gfCNCPoint4[8472] = {X 422.2320, Y 54.5599, Z -5.5000, A 0.000, B 0.000, C 0.000 }
gfCNCPoint4[8473] = {X 422.9287, Y 55.2566, Z -5.5000, A 0.000, B 0.000, C 0.000 }
gfCNCPoint4[8474] = {X 423.4529, Y 56.0909, Z -5.5000, A 0.000, B 0.000, C 0.000 }
gfCNCPoint4[8475] = {X 423.7783, Y 57.0209, Z -5.5000, A 0.000, B 0.000, C 0.000 }
gfCNCPoint4[8476] = {X 423.8886, Y 58.0000, Z -5.5000, A 0.000, B 0.000, C 0.000 }
gfCNCPoint4[8477] = {X 423.8886, Y 58.1773, Z -5.5000, A 0.000, B 0.000, C 0.000 }
gfCNCPoint4[8478] = {X 429.6420, Y 60.4190, Z -5.5000, A 0.000, B 0.000, C 0.000 }
gfCNCPoint4[8479] = {X 457.7784, Y 71.5825, Z -5.5000, A 0.000, B 0.000, C 0.000 }
gfCNCPoint4[8480] = {X 457.7788, Y 63.2811, Z -5.5000, A 0.000, B 0.000, C 0.000 }
gfCNCPoint4[8481] = {X 456.9197, Y 63.0558, Z -5.5000, A 0.000, B 0.000, C 0.000 }
gfCNCPoint4[8482] = {X 456.1233, Y 62.6625, Z -5.5000, A 0.000, B 0.000, C 0.000 }
gfCNCPoint4[8483] = {X 455.4221, Y 62.1174, Z -5.5000, A 0.000, B 0.000, C 0.000 }
gfCNCPoint4[8484] = {X 454.8446, Y 61.4425, Z -5.5000, A 0.000, B 0.000, C 0.000 }
gfCNCPoint4[8485] = {X 454.4145, Y 60.6654, Z -5.5000, A 0.000, B 0.000, C 0.000 }
gfCNCPoint4[8486] = {X 454.1492, Y 59.8177, Z -5.5000, A 0.000, B 0.000, C 0.000 }
gfCNCPoint4[8487] = {X 454.0596, Y 58.9341, Z -5.5000, A 0.000, B 0.000, C 0.000 }
gfCNCPoint4[8488] = {X 454.0596, Y 58.0000, Z -5.5000, A 0.000, B 0.000, C 0.000 }
gfCNCPoint4[8489] = {X 454.1699, Y 57.0209, Z -5.5000, A 0.000, B 0.000, C 0.000 }
gfCNCPoint4[8490] = {X 454.4953, Y 56.0909, Z -5.5000, A 0.000, B 0.000, C 0.000 }
gfCNCPoint4[8491] = {X 455.0195, Y 55.2566, Z -5.5000, A 0.000, B 0.000, C 0.000 }
gfCNCPoint4[8492] = {X 455.7162, Y 54.5599, Z -5.5000, A 0.000, B 0.000, C 0.000 }
gfCNCPoint4[8493] = {X 456.5505, Y 54.0357, Z -5.5000, A 0.000, B 0.000, C 0.000 }
gfCNCPoint4[8494] = {X 457.4805, Y 53.7103, Z -5.5000, A 0.000, B 0.000, C 0.000 }
gfCNCPoint4[8495] = {X 458.4596, Y 53.6000, Z -5.5000, A 0.000, B 0.000, C 0.000 }
gfCNCPoint4[8496] = {X 475.0000, Y 53.6000, Z -5.5000, A 0.000, B 0.000, C 0.000 }
gfCNCPoint4[8497] = {X 475.9791, Y 53.7103, Z -5.5000, A 0.000, B 0.000, C 0.000 }
gfCNCPoint4[8498] = {X 476.9091, Y 54.0357, Z -5.5000, A 0.000, B 0.000, C 0.000 }
gfCNCPoint4[8499] = {X 477.7434, Y 54.5599, Z -5.5000, A 0.000, B 0.000, C 0.000 }
gfCNCPoint4[8500] = {X 478.4401, Y 55.2566, Z -5.5000, A 0.000, B 0.000, C 0.000 }
gfCNCPoint4[8501] = {X 478.9643, Y 56.0909, Z -5.5000, A 0.000, B 0.000, C 0.000 }
gfCNCPoint4[8502] = {X 479.2897, Y 57.0209, Z -5.5000, A 0.000, B 0.000, C 0.000 }
gfCNCPoint4[8503] = {X 479.4000, Y 58.0000, Z -5.5000, A 0.000, B 0.000, C 0.000 }
gfCNCPoint4[8504] = {X 479.3998, Y 58.9704, Z -5.5000, A 0.000, B 0.000, C 0.000 }
gfCNCPoint4[8505] = {X 479.3040, Y 59.8483, Z -5.5000, A 0.000, B 0.000, C 0.000 }
gfCNCPoint4[8506] = {X 479.0347, Y 60.6893, Z -5.5000, A 0.000, B 0.000, C 0.000 }
gfCNCPoint4[8507] = {X 478.6030, Y 61.4596, Z -5.5000, A 0.000, B 0.000, C 0.000 }
gfCNCPoint4[8508] = {X 478.0261, Y 62.1282, Z -5.5000, A 0.000, B 0.000, C 0.000 }
gfCNCPoint4[8509] = {X 477.3273, Y 62.6682, Z -5.5000, A 0.000, B 0.000, C 0.000 }
gfCNCPoint4[8510] = {X 476.5348, Y 63.0577, Z -5.5000, A 0.000, B 0.000, C 0.000 }
gfCNCPoint4[8511] = {X 475.6805, Y 63.2811, Z -5.5000, A 0.000, B 0.000, C 0.000 }
gfCNCPoint4[8512] = {X 475.6809, Y 92.7040, Z -5.5000, A 0.000, B 0.000, C 0.000 }
gfCNCPoint4[8513] = {X 476.0501, Y 92.7986, Z -5.5000, A 0.000, B 0.000, C 0.000 }
gfCNCPoint4[8514] = {X 476.4143, Y 92.9108, Z -5.5000, A 0.000, B 0.000, C 0.000 }
gfCNCPoint4[8515] = {X 477.2408, Y 93.2866, Z -5.5000, A 0.000, B 0.000, C 0.000 }
gfCNCPoint4[8516] = {X 477.9718, Y 93.8249, Z -5.5000, A 0.000, B 0.000, C 0.000 }
gfCNCPoint4[8517] = {X 478.5759, Y 94.5026, Z -5.5000, A 0.000, B 0.000, C 0.000 }
gfCNCPoint4[8518] = {X 479.0270, Y 95.2905, Z -5.5000, A 0.000, B 0.000, C 0.000 }
gfCNCPoint4[8519] = {X 479.3057, Y 96.1545, Z -5.5000, A 0.000, B 0.000, C 0.000 }
gfCNCPoint4[8520] = {X 479.4000, Y 97.0575, Z -5.5000, A 0.000, B 0.000, C 0.000 }
gfCNCPoint4[8521] = {X 479.4000, Y 97.6951, Z -5.5000, A 0.000, B 0.000, C 0.000 }
gfCNCPoint4[8522] = {X 479.8800, Y 97.6951, Z -5.5000, A 0.000, B 0.000, C 0.000 }
gfCNCPoint4[8523] = {X 507.6814, Y 97.6951, Z -5.5000, A 0.000, B 0.000, C 0.000 }
gfCNCPoint4[8524] = {X 507.6814, Y 100.0951, Z -5.5000, A 0.000, B 0.000, C 0.000 }
gfCNCPoint4[8525] = {X 600.0148, Y 100.0951, Z -5.5000, A 0.000, B 0.000, C 0.000 }
gfCNCPoint4[8526] = {X 600.0672, Y 100.0698, Z -5.5000, A 0.000, B 0.000, C 0.000 }
gfCNCPoint4[8527] = {X 600.0949, Y 100.0187, Z -5.5000, A 0.000, B 0.000, C 0.000 }
gfCNCPoint4[8528] = {X 600.0966, Y 99.1432, Z -5.5000, A 0.000, B 0.000, C 0.000 }
gfCNCPoint4[8529] = {X 600.0966, Y 49.8790, Z -5.5000, A 0.000, B 0.000, C 0.000 }
gfCNCPoint4[8530] = {X 601.1112, Y 49.7518, Z -5.5000, A 0.000, B 0.000, C 0.000 }
gfCNCPoint4[8531] = {X 602.0770, Y 49.4159, Z -5.5000, A 0.000, B 0.000, C 0.000 }
gfCNCPoint4[8532] = {X 602.9516, Y 48.8862, Z -5.5000, A 0.000, B 0.000, C 0.000 }
gfCNCPoint4[8533] = {X 603.6966, Y 48.1858, Z -5.5000, A 0.000, B 0.000, C 0.000 }
gfCNCPoint4[8534] = {X 603.6966, Y 47.3864, Z -5.5000, A 0.000, B 0.000, C 0.000 }
gfCNCPoint4[8535] = {X 603.1503, Y 48.0717, Z -5.5000, A 0.000, B 0.000, C 0.000 }
gfCNCPoint4[8536] = {X 602.4791, Y 48.6351, Z -5.5000, A 0.000, B 0.000, C 0.000 }
gfCNCPoint4[8537] = {X 601.7094, Y 49.0544, Z -5.5000, A 0.000, B 0.000, C 0.000 }
gfCNCPoint4[8538] = {X 600.8720, Y 49.3127, Z -5.5000, A 0.000, B 0.000, C 0.000 }
gfCNCPoint4[8539] = {X 600.0000, Y 49.4000, Z -5.5000, A 0.000, B 0.000, C 0.000 }
gfCNCPoint4[8540] = {X 593.5565, Y 49.4000, Z -5.5000, A 0.000, B 0.000, C 0.000 }
gfCNCPoint4[8541] = {X 592.5988, Y 49.2945, Z -5.5000, A 0.000, B 0.000, C 0.000 }
gfCNCPoint4[8542] = {X 591.6870, Y 48.9831, Z -5.5000, A 0.000, B 0.000, C 0.000 }
gfCNCPoint4[8543] = {X 590.8648, Y 48.4806, Z -5.5000, A 0.000, B 0.000, C 0.000 }
gfCNCPoint4[8544] = {X 590.1717, Y 47.8112, Z -5.5000, A 0.000, B 0.000, C 0.000 }
gfCNCPoint4[8545] = {X 589.6410, Y 47.0071, Z -5.5000, A 0.000, B 0.000, C 0.000 }
gfCNCPoint4[8546] = {X 589.3741, Y 46.3664, Z -5.5000, A 0.000, B 0.000, C 0.000 }
gfCNCPoint4[8547] = {X 589.2113, Y 45.6918, Z -5.5000, A 0.000, B 0.000, C 0.000 }
gfCNCPoint4[8548] = {X 589.1565, Y 45.0000, Z -5.5000, A 0.000, B 0.000, C 0.000 }
gfCNCPoint4[8549] = {X 589.1565, Y 44.0643, Z -5.5000, A 0.000, B 0.000, C 0.000 }
gfCNCPoint4[8550] = {X 589.2606, Y 43.1278, Z -5.5000, A 0.000, B 0.000, C 0.000 }
gfCNCPoint4[8551] = {X 589.5599, Y 42.2344, Z -5.5000, A 0.000, B 0.000, C 0.000 }
gfCNCPoint4[8552] = {X 590.0411, Y 41.4243, Z -5.5000, A 0.000, B 0.000, C 0.000 }
gfCNCPoint4[8553] = {X 590.6824, Y 40.7340, Z -5.5000, A 0.000, B 0.000, C 0.000 }
gfCNCPoint4[8554] = {X 590.6838, Y 40.3070, Z -5.5000, A 0.000, B 0.000, C 0.000 }
gfCNCPoint4[8555] = {X 590.6830, Y 35.2188, Z -5.5000, A 0.000, B 0.000, C 0.000 }
gfCNCPoint4[8556] = {X 590.6828, Y 33.9412, Z -5.5000, A 0.000, B 0.000, C 0.000 }
gfCNCPoint4[8557] = {X 585.5192, Y 46.6830, Z -5.5000, A 0.000, B 0.000, C 0.000 }
gfCNCPoint4[8558] = {X 585.4476, Y 46.8466, Z -5.5000, A 0.000, B 0.000, C 0.000 }
gfCNCPoint4[8559] = {X 585.3694, Y 47.0071, Z -5.5000, A 0.000, B 0.000, C 0.000 }
gfCNCPoint4[8560] = {X 584.8417, Y 47.8075, Z -5.5000, A 0.000, B 0.000, C 0.000 }
gfCNCPoint4[8561] = {X 584.1532, Y 48.4747, Z -5.5000, A 0.000, B 0.000, C 0.000 }
gfCNCPoint4[8562] = {X 583.3365, Y 48.9769, Z -5.5000, A 0.000, B 0.000, C 0.000 }
gfCNCPoint4[8563] = {X 582.4111, Y 49.2946, Z -5.5000, A 0.000, B 0.000, C 0.000 }
gfCNCPoint4[8564] = {X 581.4384, Y 49.4000, Z -5.5000, A 0.000, B 0.000, C 0.000 }
gfCNCPoint4[8565] = {X 580.4664, Y 49.2878, Z -5.5000, A 0.000, B 0.000, C 0.000 }
gfCNCPoint4[8566] = {X 579.5433, Y 48.9635, Z -5.5000, A 0.000, B 0.000, C 0.000 }
gfCNCPoint4[8567] = {X 578.7146, Y 48.4433, Z -5.5000, A 0.000, B 0.000, C 0.000 }
gfCNCPoint4[8568] = {X 578.0214, Y 47.7529, Z -5.5000, A 0.000, B 0.000, C 0.000 }
gfCNCPoint4[8569] = {X 577.4979, Y 46.9263, Z -5.5000, A 0.000, B 0.000, C 0.000 }
gfCNCPoint4[8570] = {X 577.4375, Y 46.7968, Z -5.5000, A 0.000, B 0.000, C 0.000 }
gfCNCPoint4[8571] = {X 577.3813, Y 46.6655, Z -5.5000, A 0.000, B 0.000, C 0.000 }
gfCNCPoint4[8572] = {X 572.5793, Y 34.9232, Z -5.5000, A 0.000, B 0.000, C 0.000 }
gfCNCPoint4[8573] = {X 572.0992, Y 33.7494, Z -5.5000, A 0.000, B 0.000, C 0.000 }
gfCNCPoint4[8574] = {X 572.0993, Y 35.0176, Z -5.5000, A 0.000, B 0.000, C 0.000 }
gfCNCPoint4[8575] = {X 572.0995, Y 40.7335, Z -5.5000, A 0.000, B 0.000, C 0.000 }
gfCNCPoint4[8576] = {X 572.7439, Y 41.4225, Z -5.5000, A 0.000, B 0.000, C 0.000 }
gfCNCPoint4[8577] = {X 573.2265, Y 42.2331, Z -5.5000, A 0.000, B 0.000, C 0.000 }
gfCNCPoint4[8578] = {X 573.5253, Y 43.1280, Z -5.5000, A 0.000, B 0.000, C 0.000 }
gfCNCPoint4[8579] = {X 573.6264, Y 44.0660, Z -5.5000, A 0.000, B 0.000, C 0.000 }
gfCNCPoint4[8580] = {X 573.6264, Y 45.0000, Z -5.5000, A 0.000, B 0.000, C 0.000 }
gfCNCPoint4[8581] = {X 573.5140, Y 45.9884, Z -5.5000, A 0.000, B 0.000, C 0.000 }
gfCNCPoint4[8582] = {X 573.1824, Y 46.9263, Z -5.5000, A 0.000, B 0.000, C 0.000 }
gfCNCPoint4[8583] = {X 572.6569, Y 47.7553, Z -5.5000, A 0.000, B 0.000, C 0.000 }
gfCNCPoint4[8584] = {X 571.9608, Y 48.4472, Z -5.5000, A 0.000, B 0.000, C 0.000 }
gfCNCPoint4[8585] = {X 571.1286, Y 48.9676, Z -5.5000, A 0.000, B 0.000, C 0.000 }
gfCNCPoint4[8586] = {X 570.2018, Y 49.2905, Z -5.5000, A 0.000, B 0.000, C 0.000 }
gfCNCPoint4[8587] = {X 569.2264, Y 49.4000, Z -5.5000, A 0.000, B 0.000, C 0.000 }
gfCNCPoint4[8588] = {X 562.4443, Y 49.4000, Z -5.5000, A 0.000, B 0.000, C 0.000 }
gfCNCPoint4[8589] = {X 561.4652, Y 49.2897, Z -5.5000, A 0.000, B 0.000, C 0.000 }
gfCNCPoint4[8590] = {X 560.5352, Y 48.9643, Z -5.5000, A 0.000, B 0.000, C 0.000 }
gfCNCPoint4[8591] = {X 559.7009, Y 48.4401, Z -5.5000, A 0.000, B 0.000, C 0.000 }
gfCNCPoint4[8592] = {X 559.0042, Y 47.7434, Z -5.5000, A 0.000, B 0.000, C 0.000 }
gfCNCPoint4[8593] = {X 558.4800, Y 46.9091, Z -5.5000, A 0.000, B 0.000, C 0.000 }
gfCNCPoint4[8594] = {X 558.1546, Y 45.9791, Z -5.5000, A 0.000, B 0.000, C 0.000 }
gfCNCPoint4[8595] = {X 558.0443, Y 45.0000, Z -5.5000, A 0.000, B 0.000, C 0.000 }
gfCNCPoint4[8596] = {X 558.0443, Y 44.0644, Z -5.5000, A 0.000, B 0.000, C 0.000 }
gfCNCPoint4[8597] = {X 558.1481, Y 43.1277, Z -5.5000, A 0.000, B 0.000, C 0.000 }
gfCNCPoint4[8598] = {X 558.4477, Y 42.2341, Z -5.5000, A 0.000, B 0.000, C 0.000 }
gfCNCPoint4[8599] = {X 558.9294, Y 41.4240, Z -5.5000, A 0.000, B 0.000, C 0.000 }
gfCNCPoint4[8600] = {X 559.5715, Y 40.7340, Z -5.5000, A 0.000, B 0.000, C 0.000 }
gfCNCPoint4[8601] = {X 559.5715, Y 9.2668, Z -5.5000, A 0.000, B 0.000, C 0.000 }
gfCNCPoint4[8602] = {X 558.9270, Y 8.5777, Z -5.5000, A 0.000, B 0.000, C 0.000 }
gfCNCPoint4[8603] = {X 558.4443, Y 7.7670, Z -5.5000, A 0.000, B 0.000, C 0.000 }
gfCNCPoint4[8604] = {X 558.1454, Y 6.8720, Z -5.5000, A 0.000, B 0.000, C 0.000 }
gfCNCPoint4[8605] = {X 558.0443, Y 5.9340, Z -5.5000, A 0.000, B 0.000, C 0.000 }
gfCNCPoint4[8606] = {X 558.0443, Y 5.0000, Z -5.5000, A 0.000, B 0.000, C 0.000 }
gfCNCPoint4[8607] = {X 558.1353, Y 4.1096, Z -5.5000, A 0.000, B 0.000, C 0.000 }
gfCNCPoint4[8608] = {X 558.4046, Y 3.2561, Z -5.5000, A 0.000, B 0.000, C 0.000 }
gfCNCPoint4[8609] = {X 558.9155, Y 2.3717, Z -5.5000, A 0.000, B 0.000, C 0.000 }
gfCNCPoint4[8610] = {X 559.6166, Y 1.6289, Z -5.5000, A 0.000, B 0.000, C 0.000 }
gfCNCPoint4[8611] = {X 560.4700, Y 1.0678, Z -5.5000, A 0.000, B 0.000, C 0.000 }
gfCNCPoint4[8612] = {X 561.4298, Y 0.7185, Z -5.5000, A 0.000, B 0.000, C 0.000 }
gfCNCPoint4[8613] = {X 562.4443, Y 0.6000, Z -5.5000, A 0.000, B 0.000, C 0.000 }
gfCNCPoint4[8614] = {X 570.9376, Y 0.6000, Z -5.5000, A 0.000, B 0.000, C 0.000 }
gfCNCPoint4[8615] = {X 571.9520, Y 0.7185, Z -5.5000, A 0.000, B 0.000, C 0.000 }
gfCNCPoint4[8616] = {X 572.9118, Y 1.0678, Z -5.5000, A 0.000, B 0.000, C 0.000 }
gfCNCPoint4[8617] = {X 573.7653, Y 1.6289, Z -5.5000, A 0.000, B 0.000, C 0.000 }
gfCNCPoint4[8618] = {X 574.4663, Y 2.3717, Z -5.5000, A 0.000, B 0.000, C 0.000 }
gfCNCPoint4[8619] = {X 574.9772, Y 3.2561, Z -5.5000, A 0.000, B 0.000, C 0.000 }
gfCNCPoint4[8620] = {X 575.2465, Y 4.1096, Z -5.5000, A 0.000, B 0.000, C 0.000 }
gfCNCPoint4[8621] = {X 575.3376, Y 5.0000, Z -5.5000, A 0.000, B 0.000, C 0.000 }
gfCNCPoint4[8622] = {X 575.3372, Y 5.9910, Z -5.5000, A 0.000, B 0.000, C 0.000 }
gfCNCPoint4[8623] = {X 575.2577, Y 6.7686, Z -5.5000, A 0.000, B 0.000, C 0.000 }
gfCNCPoint4[8624] = {X 575.0418, Y 7.5199, Z -5.5000, A 0.000, B 0.000, C 0.000 }
gfCNCPoint4[8625] = {X 574.6964, Y 8.2211, Z -5.5000, A 0.000, B 0.000, C 0.000 }
gfCNCPoint4[8626] = {X 575.2866, Y 9.6566, Z -5.5000, A 0.000, B 0.000, C 0.000 }
gfCNCPoint4[8627] = {X 581.1912, Y 24.1575, Z -5.5000, A 0.000, B 0.000, C 0.000 }
gfCNCPoint4[8628] = {X 587.7569, Y 8.0998, Z -5.5000, A 0.000, B 0.000, C 0.000 }
gfCNCPoint4[8629] = {X 587.4434, Y 7.4142, Z -5.5000, A 0.000, B 0.000, C 0.000 }
gfCNCPoint4[8630] = {X 587.2515, Y 6.6851, Z -5.5000, A 0.000, B 0.000, C 0.000 }
gfCNCPoint4[8631] = {X 587.1870, Y 5.9340, Z -5.5000, A 0.000, B 0.000, C 0.000 }
gfCNCPoint4[8632] = {X 587.1870, Y 5.0000, Z -5.5000, A 0.000, B 0.000, C 0.000 }
gfCNCPoint4[8633] = {X 587.2780, Y 4.1096, Z -5.5000, A 0.000, B 0.000, C 0.000 }
gfCNCPoint4[8634] = {X 587.5473, Y 3.2561, Z -5.5000, A 0.000, B 0.000, C 0.000 }
gfCNCPoint4[8635] = {X 588.0582, Y 2.3717, Z -5.5000, A 0.000, B 0.000, C 0.000 }
gfCNCPoint4[8636] = {X 588.7592, Y 1.6289, Z -5.5000, A 0.000, B 0.000, C 0.000 }
gfCNCPoint4[8637] = {X 589.6127, Y 1.0678, Z -5.5000, A 0.000, B 0.000, C 0.000 }
gfCNCPoint4[8638] = {X 590.5725, Y 0.7185, Z -5.5000, A 0.000, B 0.000, C 0.000 }
gfCNCPoint4[8639] = {X 591.5870, Y 0.6000, Z -5.5000, A 0.000, B 0.000, C 0.000 }
gfCNCPoint4[8640] = {X 600.0000, Y 0.6000, Z -5.5000, A 0.000, B 0.000, C 0.000 }
gfCNCPoint4[8641] = {X 600.8720, Y 0.6873, Z -5.5000, A 0.000, B 0.000, C 0.000 }
gfCNCPoint4[8642] = {X 601.7094, Y 0.9456, Z -5.5000, A 0.000, B 0.000, C 0.000 }
gfCNCPoint4[8643] = {X 602.4791, Y 1.3649, Z -5.5000, A 0.000, B 0.000, C 0.000 }
gfCNCPoint4[8644] = {X 603.1503, Y 1.9283, Z -5.5000, A 0.000, B 0.000, C 0.000 }
gfCNCPoint4[8645] = {X 603.6966, Y 2.6136, Z -5.5000, A 0.000, B 0.000, C 0.000 }
gfCNCPoint4[8646] = {X 603.6966, Y 1.8142, Z -5.5000, A 0.000, B 0.000, C 0.000 }
gfCNCPoint4[8647] = {X 602.9513, Y 1.1136, Z -5.5000, A 0.000, B 0.000, C 0.000 }
gfCNCPoint4[8648] = {X 602.0763, Y 0.5838, Z -5.5000, A 0.000, B 0.000, C 0.000 }
gfCNCPoint4[8649] = {X 601.1101, Y 0.2479, Z -5.5000, A 0.000, B 0.000, C 0.000 }
gfCNCPoint4[8650] = {X 600.0952, Y 0.1209, Z -5.5000, A 0.000, B 0.000, C 0.000 }
gfCNCPoint4[8651] = {X 600.0949, Y -0.0187, Z -5.5000, A 0.000, B 0.000, C 0.000 }
gfCNCPoint4[8652] = {X 600.0672, Y -0.0698, Z -5.5000, A 0.000, B 0.000, C 0.000 }
gfCNCPoint4[8653] = {X 600.0148, Y -0.0951, Z -5.5000, A 0.000, B 0.000, C 0.000 }
gfCNCPoint4[8654] = {X 580.1328, Y -0.0951, Z -5.5000, A 0.000, B 0.000, C 0.000 }
gfCNCPoint4[8655] = {X 580.1328, Y 4.7049, Z -5.5000, A 0.000, B 0.000, C 0.000 }
gfCNCPoint4[8656] = {X 580.1364, Y 4.8524, Z -5.5000, A 0.000, B 0.000, C 0.000 }
gfCNCPoint4[8657] = {X 580.1376, Y 5.0000, Z -5.5000, A 0.000, B 0.000, C 0.000 }
gfCNCPoint4[8658] = {X 580.1376, Y 5.9339, Z -5.5000, A 0.000, B 0.000, C 0.000 }
gfCNCPoint4[8659] = {X 580.0686, Y 7.0587, Z -5.5000, A 0.000, B 0.000, C 0.000 }
gfCNCPoint4[8660] = {X 579.8626, Y 8.1666, Z -5.5000, A 0.000, B 0.000, C 0.000 }
gfCNCPoint4[8661] = {X 581.2004, Y 11.4522, Z -5.5000, A 0.000, B 0.000, C 0.000 }
gfCNCPoint4[8662] = {X 582.6183, Y 7.9844, Z -5.5000, A 0.000, B 0.000, C 0.000 }
gfCNCPoint4[8663] = {X 582.4489, Y 6.9995, Z -5.5000, A 0.000, B 0.000, C 0.000 }
gfCNCPoint4[8664] = {X 582.3872, Y 6.0020, Z -5.5000, A 0.000, B 0.000, C 0.000 }
gfCNCPoint4[8665] = {X 582.3870, Y 5.0000, Z -5.5000, A 0.000, B 0.000, C 0.000 }
gfCNCPoint4[8666] = {X 582.3881, Y 4.8524, Z -5.5000, A 0.000, B 0.000, C 0.000 }
gfCNCPoint4[8667] = {X 582.3917, Y 4.7049, Z -5.5000, A 0.000, B 0.000, C 0.000 }
gfCNCPoint4[8668] = {X 580.1328, Y 4.7049, Z -5.5000, A 0.000, B 0.000, C 0.000 }
gfCNCPoint4[8669] = {X 580.1328, Y 2.3049, Z -5.5000, A 0.000, B 0.000, C 0.000 }
gfCNCPoint4[8670] = {X 577.1807, Y 2.3049, Z -5.5000, A 0.000, B 0.000, C 0.000 }
gfCNCPoint4[8671] = {X 577.5740, Y 3.5174, Z -5.5000, A 0.000, B 0.000, C 0.000 }
gfCNCPoint4[8672] = {X 577.7341, Y 4.7819, Z -5.5000, A 0.000, B 0.000, C 0.000 }
gfCNCPoint4[8673] = {X 577.7367, Y 4.8909, Z -5.5000, A 0.000, B 0.000, C 0.000 }
gfCNCPoint4[8674] = {X 577.7376, Y 5.0000, Z -5.5000, A 0.000, B 0.000, C 0.000 }
gfCNCPoint4[8675] = {X 577.7376, Y 5.9339, Z -5.5000, A 0.000, B 0.000, C 0.000 }
gfCNCPoint4[8676] = {X 577.6318, Y 7.1284, Z -5.5000, A 0.000, B 0.000, C 0.000 }
gfCNCPoint4[8677] = {X 577.3179, Y 8.2858, Z -5.5000, A 0.000, B 0.000, C 0.000 }
gfCNCPoint4[8678] = {X 577.5058, Y 8.7427, Z -5.5000, A 0.000, B 0.000, C 0.000 }
gfCNCPoint4[8679] = {X 581.1958, Y 17.8048, Z -5.5000, A 0.000, B 0.000, C 0.000 }
gfCNCPoint4[8680] = {X 585.1515, Y 8.1305, Z -5.5000, A 0.000, B 0.000, C 0.000 }
gfCNCPoint4[8681] = {X 584.8835, Y 7.0757, Z -5.5000, A 0.000, B 0.000, C 0.000 }
gfCNCPoint4[8682] = {X 584.7872, Y 5.9916, Z -5.5000, A 0.000, B 0.000, C 0.000 }
gfCNCPoint4[8683] = {X 584.7870, Y 5.0000, Z -5.5000, A 0.000, B 0.000, C 0.000 }
gfCNCPoint4[8684] = {X 584.7878, Y 4.8909, Z -5.5000, A 0.000, B 0.000, C 0.000 }
gfCNCPoint4[8685] = {X 584.7905, Y 4.7819, Z -5.5000, A 0.000, B 0.000, C 0.000 }
gfCNCPoint4[8686] = {X 584.9506, Y 3.5174, Z -5.5000, A 0.000, B 0.000, C 0.000 }
gfCNCPoint4[8687] = {X 585.3438, Y 2.3049, Z -5.5000, A 0.000, B 0.000, C 0.000 }
gfCNCPoint4[8688] = {X 580.1328, Y 2.3049, Z -5.5000, A 0.000, B 0.000, C 0.000 }
gfCNCPoint4[8689] = {X 580.1328, Y -0.0951, Z -5.5000, A 0.000, B 0.000, C 0.000 }
gfCNCPoint4[8690] = {X 351.5673, Y -0.0951, Z -5.5000, A 0.000, B 0.000, C 0.000 }
gfCNCPoint4[8691] = {X 351.4056, Y -0.1253, Z -5.5000, A 0.000, B 0.000, C 0.000 }
gfCNCPoint4[8692] = {X 348.9089, Y -0.4718, Z -5.5000, A 0.000, B 0.000, C 0.000 }
gfCNCPoint4[8693] = {X 346.3907, Y -0.5826, Z -5.5000, A 0.000, B 0.000, C 0.000 }
gfCNCPoint4[8694] = {X 343.8732, Y -0.4566, Z -5.5000, A 0.000, B 0.000, C 0.000 }
gfCNCPoint4[8695] = {X 341.3786, Y -0.0951, Z -5.5000, A 0.000, B 0.000, C 0.000 }
gfCNCPoint4[8696] = {X -0.0148, Y -0.0951, Z -5.5000, A 0.000, B 0.000, C 0.000 }
gfCNCPoint4[8697] = {X -0.0672, Y -0.0698, Z -5.5000, A 0.000, B 0.000, C 0.000 }
gfCNCPoint4[8698] = {X -0.0949, Y -0.0187, Z -5.5000, A 0.000, B 0.000, C 0.000 }
gfCNCPoint4[8699] = {X -0.0966, Y 0.8568, Z -5.5000, A 0.000, B 0.000, C 0.000 }
gfCNCPoint4[8700] = {X -0.0966, Y 8.7891, Z -5.5000, A 0.000, B 0.000, C 0.000 }
gfCNCPoint4[8701] = {X -0.7633, Y 8.9979, Z -5.5000, A 0.000, B 0.000, C 0.000 }
gfCNCPoint4[8702] = {X -1.3934, Y 9.2998, Z -5.5000, A 0.000, B 0.000, C 0.000 }
gfCNCPoint4[8703] = {X -1.9904, Y 9.6404, Z -5.5000, A 0.000, B 0.000, C 0.000 }
gfCNCPoint4[8704] = {X -2.6455, Y 10.0884, Z -5.5000, A 0.000, B 0.000, C 0.000 }
gfCNCPoint4[8705] = {X -3.2193, Y 10.6367, Z -5.5000, A 0.000, B 0.000, C 0.000 }
gfCNCPoint4[8706] = {X -3.6966, Y 11.2707, Z -5.5000, A 0.000, B 0.000, C 0.000 }
gfCNCPoint4[8707] = {X -3.6966, Y 12.3463, Z -5.5000, A 0.000, B 0.000, C 0.000 }
gfCNCPoint4[8708] = {X -3.2333, Y 11.4385, Z -5.5000, A 0.000, B 0.000, C 0.000 }
gfCNCPoint4[8709] = {X -2.5734, Y 10.6616, Z -5.5000, A 0.000, B 0.000, C 0.000 }
gfCNCPoint4[8710] = {X -1.7526, Y 10.0573, Z -5.5000, A 0.000, B 0.000, C 0.000 }
gfCNCPoint4[8711] = {X -1.0994, Y 9.6852, Z -5.5000, A 0.000, B 0.000, C 0.000 }
gfCNCPoint4[8712] = {X -0.3665, Y 9.3642, Z -5.5000, A 0.000, B 0.000, C 0.000 }
gfCNCPoint4[8713] = {X 0.4125, Y 9.1813, Z -5.5000, A 0.000, B 0.000, C 0.000 }
gfCNCPoint4[8714] = {X 1.1338, Y 9.1398, Z -5.5000, A 0.000, B 0.000, C 0.000 }
gfCNCPoint4[8715] = {X 1.8522, Y 9.2169, Z -5.5000, A 0.000, B 0.000, C 0.000 }
gfCNCPoint4[8716] = {X 2.2340, Y 9.3079, Z -5.5000, A 0.000, B 0.000, C 0.000 }
gfCNCPoint4[8717] = {X 2.6063, Y 9.4325, Z -5.5000, A 0.000, B 0.000, C 0.000 }
gfCNCPoint4[8718] = {X 3.3755, Y 9.0666, Z -5.5000, A 0.000, B 0.000, C 0.000 }
gfCNCPoint4[8719] = {X 4.1727, Y 8.7667, Z -5.5000, A 0.000, B 0.000, C 0.000 }
gfCNCPoint4[8720] = {X 6.0895, Y 8.0965, Z -5.5000, A 0.000, B 0.000, C 0.000 }
gfCNCPoint4[8721] = {X 8.0569, Y 7.5940, Z -5.5000, A 0.000, B 0.000, C 0.000 }
gfCNCPoint4[8722] = {X 10.0603, Y 7.2629, Z -5.5000, A 0.000, B 0.000, C 0.000 }
gfCNCPoint4[8723] = {X 12.0848, Y 7.1057, Z -5.5000, A 0.000, B 0.000, C 0.000 }
gfCNCPoint4[8724] = {X 14.1153, Y 7.1234, Z -5.5000, A 0.000, B 0.000, C 0.000 }
gfCNCPoint4[8725] = {X 16.1367, Y 7.3160, Z -5.5000, A 0.000, B 0.000, C 0.000 }
gfCNCPoint4[8726] = {X 16.5424, Y 7.3732, Z -5.5000, A 0.000, B 0.000, C 0.000 }
gfCNCPoint4[8727] = {X 18.2863, Y 7.7304, Z -5.5000, A 0.000, B 0.000, C 0.000 }
gfCNCPoint4[8728] = {X 19.9848, Y 8.2626, Z -5.5000, A 0.000, B 0.000, C 0.000 }
gfCNCPoint4[8729] = {X 21.6207, Y 8.9644, Z -5.5000, A 0.000, B 0.000, C 0.000 }
gfCNCPoint4[8730] = {X 23.1770, Y 9.8284, Z -5.5000, A 0.000, B 0.000, C 0.000 }
gfCNCPoint4[8731] = {X 24.6376, Y 10.8457, Z -5.5000, A 0.000, B 0.000, C 0.000 }
gfCNCPoint4[8732] = {X 25.7301, Y 11.8012, Z -5.5000, A 0.000, B 0.000, C 0.000 }
gfCNCPoint4[8733] = {X 26.7100, Y 12.8718, Z -5.5000, A 0.000, B 0.000, C 0.000 }
gfCNCPoint4[8734] = {X 27.5653, Y 14.0444, Z -5.5000, A 0.000, B 0.000, C 0.000 }
gfCNCPoint4[8735] = {X 28.2853, Y 15.3045, Z -5.5000, A 0.000, B 0.000, C 0.000 }
gfCNCPoint4[8736] = {X 28.8614, Y 16.6367, Z -5.5000, A 0.000, B 0.000, C 0.000 }
gfCNCPoint4[8737] = {X 29.3383, Y 18.3011, Z -5.5000, A 0.000, B 0.000, C 0.000 }
gfCNCPoint4[8738] = {X 29.6213, Y 20.0093, Z -5.5000, A 0.000, B 0.000, C 0.000 }
gfCNCPoint4[8739] = {X 29.7065, Y 21.7387, Z -5.5000, A 0.000, B 0.000, C 0.000 }
gfCNCPoint4[8740] = {X 29.5928, Y 23.4664, Z -5.5000, A 0.000, B 0.000, C 0.000 }
gfCNCPoint4[8741] = {X 29.2818, Y 25.1697, Z -5.5000, A 0.000, B 0.000, C 0.000 }
gfCNCPoint4[8742] = {X 28.7904, Y 26.7455, Z -5.5000, A 0.000, B 0.000, C 0.000 }
gfCNCPoint4[8743] = {X 28.0834, Y 28.2371, Z -5.5000, A 0.000, B 0.000, C 0.000 }
gfCNCPoint4[8744] = {X 27.1747, Y 29.6151, Z -5.5000, A 0.000, B 0.000, C 0.000 }
gfCNCPoint4[8745] = {X 26.3577, Y 30.5722, Z -5.5000, A 0.000, B 0.000, C 0.000 }
gfCNCPoint4[8746] = {X 25.4431, Y 31.4367, Z -5.5000, A 0.000, B 0.000, C 0.000 }
gfCNCPoint4[8747] = {X 26.1251, Y 31.7404, Z -5.5000, A 0.000, B 0.000, C 0.000 }
gfCNCPoint4[8748] = {X 26.7459, Y 32.1551, Z -5.5000, A 0.000, B 0.000, C 0.000 }
gfCNCPoint4[8749] = {X 27.2877, Y 32.6688, Z -5.5000, A 0.000, B 0.000, C 0.000 }
gfCNCPoint4[8750] = {X 27.6591, Y 33.1494, Z -5.5000, A 0.000, B 0.000, C 0.000 }
gfCNCPoint4[8751] = {X 27.9609, Y 33.6765, Z -5.5000, A 0.000, B 0.000, C 0.000 }
gfCNCPoint4[8752] = {X 30.9820, Y 39.9182, Z -5.5000, A 0.000, B 0.000, C 0.000 }
gfCNCPoint4[8753] = {X 31.3085, Y 40.8441, Z -5.5000, A 0.000, B 0.000, C 0.000 }
gfCNCPoint4[8754] = {X 31.4215, Y 41.8194, Z -5.5000, A 0.000, B 0.000, C 0.000 }
gfCNCPoint4[8755] = {X 31.3155, Y 42.7955, Z -5.5000, A 0.000, B 0.000, C 0.000 }
gfCNCPoint4[8756] = {X 30.9956, Y 43.7238, Z -5.5000, A 0.000, B 0.000, C 0.000 }
gfCNCPoint4[8757] = {X 30.4779, Y 44.5580, Z -5.5000, A 0.000, B 0.000, C 0.000 }
gfCNCPoint4[8758] = {X 29.7880, Y 45.2567, Z -5.5000, A 0.000, B 0.000, C 0.000 }
gfCNCPoint4[8759] = {X 29.2519, Y 45.6902, Z -5.5000, A 0.000, B 0.000, C 0.000 }
gfCNCPoint4[8760] = {X 28.5410, Y 46.1590, Z -5.5000, A 0.000, B 0.000, C 0.000 }
gfCNCPoint4[8761] = {X 27.7532, Y 46.4826, Z -5.5000, A 0.000, B 0.000, C 0.000 }
gfCNCPoint4[8762] = {X 26.9179, Y 46.6488, Z -5.5000, A 0.000, B 0.000, C 0.000 }
gfCNCPoint4[8763] = {X 26.0663, Y 46.6515, Z -5.5000, A 0.000, B 0.000, C 0.000 }
gfCNCPoint4[8764] = {X 25.2300, Y 46.4905, Z -5.5000, A 0.000, B 0.000, C 0.000 }
gfCNCPoint4[8765] = {X 23.4344, Y 47.4362, Z -5.5000, A 0.000, B 0.000, C 0.000 }
gfCNCPoint4[8766] = {X 21.5775, Y 48.2552, Z -5.5000, A 0.000, B 0.000, C 0.000 }
gfCNCPoint4[8767] = {X 19.6684, Y 48.9436, Z -5.5000, A 0.000, B 0.000, C 0.000 }
gfCNCPoint4[8768] = {X 19.5108, Y 48.9961, Z -5.5000, A 0.000, B 0.000, C 0.000 }
gfCNCPoint4[8769] = {X 17.5871, Y 49.5249, Z -5.5000, A 0.000, B 0.000, C 0.000 }
gfCNCPoint4[8770] = {X 15.6247, Y 49.8838, Z -5.5000, A 0.000, B 0.000, C 0.000 }
gfCNCPoint4[8771] = {X 13.6384, Y 50.0702, Z -5.5000, A 0.000, B 0.000, C 0.000 }
gfCNCPoint4[8772] = {X 11.6434, Y 50.0826, Z -5.5000, A 0.000, B 0.000, C 0.000 }
gfCNCPoint4[8773] = {X 9.6550, Y 49.9208, Z -5.5000, A 0.000, B 0.000, C 0.000 }
gfCNCPoint4[8774] = {X 7.6883, Y 49.5862, Z -5.5000, A 0.000, B 0.000, C 0.000 }
gfCNCPoint4[8775] = {X 6.2183, Y 49.2055, Z -5.5000, A 0.000, B 0.000, C 0.000 }
gfCNCPoint4[8776] = {X 4.7887, Y 48.6934, Z -5.5000, A 0.000, B 0.000, C 0.000 }
gfCNCPoint4[8777] = {X 3.4113, Y 48.0540, Z -5.5000, A 0.000, B 0.000, C 0.000 }
gfCNCPoint4[8778] = {X 1.9574, Y 47.2020, Z -5.5000, A 0.000, B 0.000, C 0.000 }
gfCNCPoint4[8779] = {X 0.5963, Y 46.2083, Z -5.5000, A 0.000, B 0.000, C 0.000 }
gfCNCPoint4[8780] = {X -0.5429, Y 45.1842, Z -5.5000, A 0.000, B 0.000, C 0.000 }
gfCNCPoint4[8781] = {X -1.5547, Y 44.0340, Z -5.5000, A 0.000, B 0.000, C 0.000 }
gfCNCPoint4[8782] = {X -2.4252, Y 42.7735, Z -5.5000, A 0.000, B 0.000, C 0.000 }
gfCNCPoint4[8783] = {X -3.1424, Y 41.4199, Z -5.5000, A 0.000, B 0.000, C 0.000 }
gfCNCPoint4[8784] = {X -3.6966, Y 39.9918, Z -5.5000, A 0.000, B 0.000, C 0.000 }
gfCNCPoint4[8785] = {X -3.6966, Y 41.3546, Z -5.5000, A 0.000, B 0.000, C 0.000 }
gfCNCPoint4[8786] = {X -3.0108, Y 42.7254, Z -5.5000, A 0.000, B 0.000, C 0.000 }
gfCNCPoint4[8787] = {X -2.1748, Y 44.0101, Z -5.5000, A 0.000, B 0.000, C 0.000 }
gfCNCPoint4[8788] = {X -1.1993, Y 45.1924, Z -5.5000, A 0.000, B 0.000, C 0.000 }
gfCNCPoint4[8789] = {X -0.0966, Y 46.2571, Z -5.5000, A 0.000, B 0.000, C 0.000 }
gfCNCPoint4[8790] = {X -0.0966, Y 99.1432, Z -5.5000, A 0.000, B 0.000, C 0.000 }
gfCNCPoint4[8791] = {X -0.0949, Y 100.0187, Z -5.5000, A 0.000, B 0.000, C 0.000 }
gfCNCPoint4[8792] = {X -0.0672, Y 100.0698, Z -5.5000, A 0.000, B 0.000, C 0.000 }
gfCNCPoint4[8793] = {X -0.0148, Y 100.0951, Z -5.5000, A 0.000, B 0.000, C 0.000 }
gfCNCPoint4[8794] = {X 120.5926, Y 100.0951, Z -5.5000, A 0.000, B 0.000, C 0.000 }
gfCNCPoint4[8795] = {X 121.0614, Y 100.8812, Z -5.5000, A 0.000, B 0.000, C 0.000 }
gfCNCPoint4[8796] = {X 121.6687, Y 101.5661, Z -5.5000, A 0.000, B 0.000, C 0.000 }
gfCNCPoint4[8797] = {X 122.3932, Y 102.1254, Z -5.5000, A 0.000, B 0.000, C 0.000 }
gfCNCPoint4[8798] = {X 123.2095, Y 102.5396, Z -5.5000, A 0.000, B 0.000, C 0.000 }
gfCNCPoint4[8799] = {X 124.0887, Y 102.7942, Z -5.5000, A 0.000, B 0.000, C 0.000 }
gfCNCPoint4[8800] = {X 125.0000, Y 102.8800, Z -5.5000, A 0.000, B 0.000, C 0.000 }
gfCNCPoint4[8801] = {X 143.7791, Y 102.8800, Z -5.5000, A 0.000, B 0.000, C 0.000 }
gfCNCPoint4[8802] = {X 144.6904, Y 102.7942, Z -5.5000, A 0.000, B 0.000, C 0.000 }
gfCNCPoint4[8803] = {X 145.5696, Y 102.5396, Z -5.5000, A 0.000, B 0.000, C 0.000 }
gfCNCPoint4[8804] = {X 146.3859, Y 102.1254, Z -5.5000, A 0.000, B 0.000, C 0.000 }
gfCNCPoint4[8805] = {X 147.1104, Y 101.5661, Z -5.5000, A 0.000, B 0.000, C 0.000 }
gfCNCPoint4[8806] = {X 147.7177, Y 100.8812, Z -5.5000, A 0.000, B 0.000, C 0.000 }
gfCNCPoint4[8807] = {X 148.1865, Y 100.0951, Z -5.5000, A 0.000, B 0.000, C 0.000 }
gfCNCPoint4[8808] = {X 150.8379, Y 100.0951, Z -5.5000, A 0.000, B 0.000, C 0.000 }
gfCNCPoint4[8809] = {X 150.8379, Y 95.2951, Z -5.5000, A 0.000, B 0.000, C 0.000 }
gfCNCPoint4[8810] = {X 187.9256, Y 95.2951, Z -5.5000, A 0.000, B 0.000, C 0.000 }
gfCNCPoint4[8811] = {X 187.9777, Y 95.0990, Z -5.5000, A 0.000, B 0.000, C 0.000 }
gfCNCPoint4[8812] = {X 188.0352, Y 94.9045, Z -5.5000, A 0.000, B 0.000, C 0.000 }
gfCNCPoint4[8813] = {X 187.2619, Y 94.0602, Z -5.5000, A 0.000, B 0.000, C 0.000 }
gfCNCPoint4[8814] = {X 151.4055, Y 94.0602, Z -5.5000, A 0.000, B 0.000, C 0.000 }
gfCNCPoint4[8815] = {X 150.7059, Y 94.8353, Z -5.5000, A 0.000, B 0.000, C 0.000 }
gfCNCPoint4[8816] = {X 150.7757, Y 95.0641, Z -5.5000, A 0.000, B 0.000, C 0.000 }
gfCNCPoint4[8817] = {X 150.8379, Y 95.2951, Z -5.5000, A 0.000, B 0.000, C 0.000 }
gfCNCPoint4[8818] = {X 150.8379, Y 97.6951, Z -5.5000, A 0.000, B 0.000, C 0.000 }
gfCNCPoint4[8819] = {X 190.1070, Y 97.6951, Z -5.5000, A 0.000, B 0.000, C 0.000 }
gfCNCPoint4[8820] = {X 190.1070, Y 97.0659, Z -5.5000, A 0.000, B 0.000, C 0.000 }
gfCNCPoint4[8821] = {X 190.1938, Y 96.1495, Z -5.5000, A 0.000, B 0.000, C 0.000 }
gfCNCPoint4[8822] = {X 190.4511, Y 95.2657, Z -5.5000, A 0.000, B 0.000, C 0.000 }
gfCNCPoint4[8823] = {X 190.8699, Y 94.4460, Z -5.5000, A 0.000, B 0.000, C 0.000 }
gfCNCPoint4[8824] = {X 188.3182, Y 91.6602, Z -5.5000, A 0.000, B 0.000, C 0.000 }
gfCNCPoint4[8825] = {X 150.3387, Y 91.6602, Z -5.5000, A 0.000, B 0.000, C 0.000 }
gfCNCPoint4[8826] = {X 147.8640, Y 94.4019, Z -5.5000, A 0.000, B 0.000, C 0.000 }
gfCNCPoint4[8827] = {X 148.2982, Y 95.2325, Z -5.5000, A 0.000, B 0.000, C 0.000 }
gfCNCPoint4[8828] = {X 148.5665, Y 96.1305, Z -5.5000, A 0.000, B 0.000, C 0.000 }
gfCNCPoint4[8829] = {X 148.6591, Y 97.0632, Z -5.5000, A 0.000, B 0.000, C 0.000 }
gfCNCPoint4[8830] = {X 148.6591, Y 97.6951, Z -5.5000, A 0.000, B 0.000, C 0.000 }
gfCNCPoint4[8831] = {X 150.8379, Y 97.6951, Z -5.5000, A 0.000, B 0.000, C 0.000 }
gfCNCPoint4[8832] = {X 150.8379, Y 100.0951, Z -5.5000, A 0.000, B 0.000, C 0.000 }
gfCNCPoint4[8833] = {X 190.5796, Y 100.0951, Z -5.5000, A 0.000, B 0.000, C 0.000 }
gfCNCPoint4[8834] = {X 191.0483, Y 100.8812, Z -5.5000, A 0.000, B 0.000, C 0.000 }
gfCNCPoint4[8835] = {X 191.6557, Y 101.5661, Z -5.5000, A 0.000, B 0.000, C 0.000 }
gfCNCPoint4[8836] = {X 192.3802, Y 102.1254, Z -5.5000, A 0.000, B 0.000, C 0.000 }
gfCNCPoint4[8837] = {X 193.1964, Y 102.5396, Z -5.5000, A 0.000, B 0.000, C 0.000 }
gfCNCPoint4[8838] = {X 194.0757, Y 102.7942, Z -5.5000, A 0.000, B 0.000, C 0.000 }
gfCNCPoint4[8839] = {X 194.9870, Y 102.8800, Z -5.5000, A 0.000, B 0.000, C 0.000 }
gfCNCPoint4[8840] = {X 212.6141, Y 102.8800, Z -5.5000, A 0.000, B 0.000, C 0.000 }
gfCNCPoint4[8841] = {X 213.0066, Y 102.8642, Z -5.5000, A 0.000, B 0.000, C 0.000 }
gfCNCPoint4[8842] = {X 213.3966, Y 102.8169, Z -5.5000, A 0.000, B 0.000, C 0.000 }
gfCNCPoint4[8843] = {X 213.7865, Y 102.8642, Z -5.5000, A 0.000, B 0.000, C 0.000 }
gfCNCPoint4[8844] = {X 214.1790, Y 102.8800, Z -5.5000, A 0.000, B 0.000, C 0.000 }
gfCNCPoint4[8845] = {X 233.4798, Y 102.8800, Z -5.5000, A 0.000, B 0.000, C 0.000 }
gfCNCPoint4[8846] = {X 234.3911, Y 102.7942, Z -5.5000, A 0.000, B 0.000, C 0.000 }
gfCNCPoint4[8847] = {X 235.2703, Y 102.5396, Z -5.5000, A 0.000, B 0.000, C 0.000 }
gfCNCPoint4[8848] = {X 236.0866, Y 102.1254, Z -5.5000, A 0.000, B 0.000, C 0.000 }
gfCNCPoint4[8849] = {X 236.8111, Y 101.5661, Z -5.5000, A 0.000, B 0.000, C 0.000 }
gfCNCPoint4[8850] = {X 237.4184, Y 100.8812, Z -5.5000, A 0.000, B 0.000, C 0.000 }
gfCNCPoint4[8851] = {X 237.8872, Y 100.0951, Z -5.5000, A 0.000, B 0.000, C 0.000 }
gfCNCPoint4[8852] = {X 261.4779, Y 100.0951, Z -5.5000, A 0.000, B 0.000, C 0.000 }
gfCNCPoint4[8853] = {X 261.4779, Y 90.4951, Z -5.5000, A 0.000, B 0.000, C 0.000 }
gfCNCPoint4[8854] = {X 266.0961, Y 90.4951, Z -5.5000, A 0.000, B 0.000, C 0.000 }
gfCNCPoint4[8855] = {X 266.1752, Y 90.3747, Z -5.5000, A 0.000, B 0.000, C 0.000 }
gfCNCPoint4[8856] = {X 266.2556, Y 90.2554, Z -5.5000, A 0.000, B 0.000, C 0.000 }
gfCNCPoint4[8857] = {X 263.5098, Y 89.1790, Z -5.5000, A 0.000, B 0.000, C 0.000 }
gfCNCPoint4[8858] = {X 261.4779, Y 90.4951, Z -5.5000, A 0.000, B 0.000, C 0.000 }
gfCNCPoint4[8859] = {X 261.4779, Y 92.8951, Z -5.5000, A 0.000, B 0.000, C 0.000 }
gfCNCPoint4[8860] = {X 267.4974, Y 92.8951, Z -5.5000, A 0.000, B 0.000, C 0.000 }
gfCNCPoint4[8861] = {X 267.8429, Y 92.2375, Z -5.5000, A 0.000, B 0.000, C 0.000 }
gfCNCPoint4[8862] = {X 268.2378, Y 91.6085, Z -5.5000, A 0.000, B 0.000, C 0.000 }
gfCNCPoint4[8863] = {X 269.1700, Y 90.4463, Z -5.5000, A 0.000, B 0.000, C 0.000 }
gfCNCPoint4[8864] = {X 270.2694, Y 89.4409, Z -5.5000, A 0.000, B 0.000, C 0.000 }
gfCNCPoint4[8865] = {X 270.2694, Y 89.2510, Z -5.5000, A 0.000, B 0.000, C 0.000 }
gfCNCPoint4[8866] = {X 263.2389, Y 86.4950, Z -5.5000, A 0.000, B 0.000, C 0.000 }
gfCNCPoint4[8867] = {X 253.3580, Y 92.8951, Z -5.5000, A 0.000, B 0.000, C 0.000 }
gfCNCPoint4[8868] = {X 261.4779, Y 92.8951, Z -5.5000, A 0.000, B 0.000, C 0.000 }
gfCNCPoint4[8869] = {X 261.4779, Y 95.2951, Z -5.5000, A 0.000, B 0.000, C 0.000 }
gfCNCPoint4[8870] = {X 269.1714, Y 95.2951, Z -5.5000, A 0.000, B 0.000, C 0.000 }
gfCNCPoint4[8871] = {X 269.5515, Y 94.1745, Z -5.5000, A 0.000, B 0.000, C 0.000 }
gfCNCPoint4[8872] = {X 270.1082, Y 93.1303, Z -5.5000, A 0.000, B 0.000, C 0.000 }
gfCNCPoint4[8873] = {X 270.8267, Y 92.1901, Z -5.5000, A 0.000, B 0.000, C 0.000 }
gfCNCPoint4[8874] = {X 271.6880, Y 91.3787, Z -5.5000, A 0.000, B 0.000, C 0.000 }
gfCNCPoint4[8875] = {X 272.6694, Y 90.7176, Z -5.5000, A 0.000, B 0.000, C 0.000 }
gfCNCPoint4[8876] = {X 272.6694, Y 87.6139, Z -5.5000, A 0.000, B 0.000, C 0.000 }
gfCNCPoint4[8877] = {X 262.9680, Y 83.8110, Z -5.5000, A 0.000, B 0.000, C 0.000 }
gfCNCPoint4[8878] = {X 245.2381, Y 95.2951, Z -5.5000, A 0.000, B 0.000, C 0.000 }
gfCNCPoint4[8879] = {X 261.4779, Y 95.2951, Z -5.5000, A 0.000, B 0.000, C 0.000 }
gfCNCPoint4[8880] = {X 261.4779, Y 97.6951, Z -5.5000, A 0.000, B 0.000, C 0.000 }
gfCNCPoint4[8881] = {X 271.3527, Y 97.6951, Z -5.5000, A 0.000, B 0.000, C 0.000 }
gfCNCPoint4[8882] = {X 271.3529, Y 97.0186, Z -5.5000, A 0.000, B 0.000, C 0.000 }
gfCNCPoint4[8883] = {X 271.4810, Y 95.9545, Z -5.5000, A 0.000, B 0.000, C 0.000 }
gfCNCPoint4[8884] = {X 271.8382, Y 94.9440, Z -5.5000, A 0.000, B 0.000, C 0.000 }
gfCNCPoint4[8885] = {X 272.4073, Y 94.0359, Z -5.5000, A 0.000, B 0.000, C 0.000 }
gfCNCPoint4[8886] = {X 273.1610, Y 93.2739, Z -5.5000, A 0.000, B 0.000, C 0.000 }
gfCNCPoint4[8887] = {X 274.0629, Y 92.6949, Z -5.5000, A 0.000, B 0.000, C 0.000 }
gfCNCPoint4[8888] = {X 275.0694, Y 92.3266, Z -5.5000, A 0.000, B 0.000, C 0.000 }
gfCNCPoint4[8889] = {X 275.0694, Y 85.9769, Z -5.5000, A 0.000, B 0.000, C 0.000 }
gfCNCPoint4[8890] = {X 262.6990, Y 81.1277, Z -5.5000, A 0.000, B 0.000, C 0.000 }
gfCNCPoint4[8891] = {X 262.5791, Y 81.2034, Z -5.5000, A 0.000, B 0.000, C 0.000 }
gfCNCPoint4[8892] = {X 238.3587, Y 96.8915, Z -5.5000, A 0.000, B 0.000, C 0.000 }
gfCNCPoint4[8893] = {X 238.3598, Y 97.0659, Z -5.5000, A 0.000, B 0.000, C 0.000 }
gfCNCPoint4[8894] = {X 238.3598, Y 97.6951, Z -5.5000, A 0.000, B 0.000, C 0.000 }
gfCNCPoint4[8895] = {X 261.4779, Y 97.6951, Z -5.5000, A 0.000, B 0.000, C 0.000 }
gfCNCPoint4[8896] = {X 261.4779, Y 100.0951, Z -5.5000, A 0.000, B 0.000, C 0.000 }
gfCNCPoint4[8897] = {X 271.8253, Y 100.0951, Z -5.5000, A 0.000, B 0.000, C 0.000 }
gfCNCPoint4[8898] = {X 272.2941, Y 100.8812, Z -5.5000, A 0.000, B 0.000, C 0.000 }
gfCNCPoint4[8899] = {X 272.9014, Y 101.5661, Z -5.5000, A 0.000, B 0.000, C 0.000 }
gfCNCPoint4[8900] = {X 273.6259, Y 102.1254, Z -5.5000, A 0.000, B 0.000, C 0.000 }
gfCNCPoint4[8901] = {X 274.4422, Y 102.5396, Z -5.5000, A 0.000, B 0.000, C 0.000 }
gfCNCPoint4[8902] = {X 275.3214, Y 102.7942, Z -5.5000, A 0.000, B 0.000, C 0.000 }
gfCNCPoint4[8903] = {X 276.2327, Y 102.8800, Z -5.5000, A 0.000, B 0.000, C 0.000 }
gfCNCPoint4[8904] = {X 292.7731, Y 102.8800, Z -5.5000, A 0.000, B 0.000, C 0.000 }
gfCNCPoint4[8905] = {X 293.6844, Y 102.7942, Z -5.5000, A 0.000, B 0.000, C 0.000 }
gfCNCPoint4[8906] = {X 294.5636, Y 102.5396, Z -5.5000, A 0.000, B 0.000, C 0.000 }
gfCNCPoint4[8907] = {X 295.3799, Y 102.1254, Z -5.5000, A 0.000, B 0.000, C 0.000 }
gfCNCPoint4[8908] = {X 296.1044, Y 101.5661, Z -5.5000, A 0.000, B 0.000, C 0.000 }
gfCNCPoint4[8909] = {X 296.7117, Y 100.8812, Z -5.5000, A 0.000, B 0.000, C 0.000 }
gfCNCPoint4[8910] = {X 297.1805, Y 100.0951, Z -5.5000, A 0.000, B 0.000, C 0.000 }
gfCNCPoint4[8911] = {X 319.1327, Y 100.0951, Z -5.5000, A 0.000, B 0.000, C 0.000 }
gfCNCPoint4[8912] = {X 321.4362, Y 100.8684, Z -5.5000, A 0.000, B 0.000, C 0.000 }
gfCNCPoint4[8913] = {X 323.7824, Y 101.5005, Z -5.5000, A 0.000, B 0.000, C 0.000 }
gfCNCPoint4[8914] = {X 326.1626, Y 101.9890, Z -5.5000, A 0.000, B 0.000, C 0.000 }
gfCNCPoint4[8915] = {X 330.1025, Y 102.5984, Z -5.5000, A 0.000, B 0.000, C 0.000 }
gfCNCPoint4[8916] = {X 334.0644, Y 103.0428, Z -5.5000, A 0.000, B 0.000, C 0.000 }
gfCNCPoint4[8917] = {X 338.0414, Y 103.3214, Z -5.5000, A 0.000, B 0.000, C 0.000 }
gfCNCPoint4[8918] = {X 343.7798, Y 103.5420, Z -5.5000, A 0.000, B 0.000, C 0.000 }
gfCNCPoint4[8919] = {X 349.5224, Y 103.5871, Z -5.5000, A 0.000, B 0.000, C 0.000 }
gfCNCPoint4[8920] = {X 355.2636, Y 103.4567, Z -5.5000, A 0.000, B 0.000, C 0.000 }
gfCNCPoint4[8921] = {X 360.9982, Y 103.1509, Z -5.5000, A 0.000, B 0.000, C 0.000 }
gfCNCPoint4[8922] = {X 364.9924, Y 102.7831, Z -5.5000, A 0.000, B 0.000, C 0.000 }
gfCNCPoint4[8923] = {X 368.9636, Y 102.2187, Z -5.5000, A 0.000, B 0.000, C 0.000 }
gfCNCPoint4[8924] = {X 372.9022, Y 101.4592, Z -5.5000, A 0.000, B 0.000, C 0.000 }
gfCNCPoint4[8925] = {X 375.2293, Y 100.8562, Z -5.5000, A 0.000, B 0.000, C 0.000 }
gfCNCPoint4[8926] = {X 377.5096, Y 100.0951, Z -5.5000, A 0.000, B 0.000, C 0.000 }
gfCNCPoint4[8927] = {X 391.9986, Y 100.0951, Z -5.5000, A 0.000, B 0.000, C 0.000 }
gfCNCPoint4[8928] = {X 392.4673, Y 100.8812, Z -5.5000, A 0.000, B 0.000, C 0.000 }
gfCNCPoint4[8929] = {X 393.0747, Y 101.5661, Z -5.5000, A 0.000, B 0.000, C 0.000 }
gfCNCPoint4[8930] = {X 393.7992, Y 102.1254, Z -5.5000, A 0.000, B 0.000, C 0.000 }
gfCNCPoint4[8931] = {X 394.6154, Y 102.5396, Z -5.5000, A 0.000, B 0.000, C 0.000 }
gfCNCPoint4[8932] = {X 395.4947, Y 102.7942, Z -5.5000, A 0.000, B 0.000, C 0.000 }
gfCNCPoint4[8933] = {X 396.4059, Y 102.8800, Z -5.5000, A 0.000, B 0.000, C 0.000 }
gfCNCPoint4[8934] = {X 415.7067, Y 102.8800, Z -5.5000, A 0.000, B 0.000, C 0.000 }
gfCNCPoint4[8935] = {X 416.6180, Y 102.7942, Z -5.5000, A 0.000, B 0.000, C 0.000 }
gfCNCPoint4[8936] = {X 417.4972, Y 102.5396, Z -5.5000, A 0.000, B 0.000, C 0.000 }
gfCNCPoint4[8937] = {X 418.3135, Y 102.1254, Z -5.5000, A 0.000, B 0.000, C 0.000 }
gfCNCPoint4[8938] = {X 419.0380, Y 101.5661, Z -5.5000, A 0.000, B 0.000, C 0.000 }
gfCNCPoint4[8939] = {X 419.6453, Y 100.8812, Z -5.5000, A 0.000, B 0.000, C 0.000 }
gfCNCPoint4[8940] = {X 420.1141, Y 100.0951, Z -5.5000, A 0.000, B 0.000, C 0.000 }
gfCNCPoint4[8941] = {X 443.7032, Y 100.0951, Z -5.5000, A 0.000, B 0.000, C 0.000 }
gfCNCPoint4[8942] = {X 443.7032, Y 90.4951, Z -5.5000, A 0.000, B 0.000, C 0.000 }
gfCNCPoint4[8943] = {X 448.3230, Y 90.4951, Z -5.5000, A 0.000, B 0.000, C 0.000 }
gfCNCPoint4[8944] = {X 448.4021, Y 90.3747, Z -5.5000, A 0.000, B 0.000, C 0.000 }
gfCNCPoint4[8945] = {X 448.4825, Y 90.2554, Z -5.5000, A 0.000, B 0.000, C 0.000 }
gfCNCPoint4[8946] = {X 445.7356, Y 89.1786, Z -5.5000, A 0.000, B 0.000, C 0.000 }
gfCNCPoint4[8947] = {X 443.7032, Y 90.4951, Z -5.5000, A 0.000, B 0.000, C 0.000 }
gfCNCPoint4[8948] = {X 443.7032, Y 92.8951, Z -5.5000, A 0.000, B 0.000, C 0.000 }
gfCNCPoint4[8949] = {X 449.7243, Y 92.8951, Z -5.5000, A 0.000, B 0.000, C 0.000 }
gfCNCPoint4[8950] = {X 450.0698, Y 92.2375, Z -5.5000, A 0.000, B 0.000, C 0.000 }
gfCNCPoint4[8951] = {X 450.4647, Y 91.6084, Z -5.5000, A 0.000, B 0.000, C 0.000 }
gfCNCPoint4[8952] = {X 451.3969, Y 90.4463, Z -5.5000, A 0.000, B 0.000, C 0.000 }
gfCNCPoint4[8953] = {X 452.4963, Y 89.4409, Z -5.5000, A 0.000, B 0.000, C 0.000 }
gfCNCPoint4[8954] = {X 452.4963, Y 89.2510, Z -5.5000, A 0.000, B 0.000, C 0.000 }
gfCNCPoint4[8955] = {X 445.4646, Y 86.4945, Z -5.5000, A 0.000, B 0.000, C 0.000 }
gfCNCPoint4[8956] = {X 435.5839, Y 92.8951, Z -5.5000, A 0.000, B 0.000, C 0.000 }
gfCNCPoint4[8957] = {X 443.7032, Y 92.8951, Z -5.5000, A 0.000, B 0.000, C 0.000 }
gfCNCPoint4[8958] = {X 443.7032, Y 95.2951, Z -5.5000, A 0.000, B 0.000, C 0.000 }
gfCNCPoint4[8959] = {X 451.3983, Y 95.2951, Z -5.5000, A 0.000, B 0.000, C 0.000 }
gfCNCPoint4[8960] = {X 451.7784, Y 94.1745, Z -5.5000, A 0.000, B 0.000, C 0.000 }
gfCNCPoint4[8961] = {X 452.3351, Y 93.1303, Z -5.5000, A 0.000, B 0.000, C 0.000 }
gfCNCPoint4[8962] = {X 453.0536, Y 92.1901, Z -5.5000, A 0.000, B 0.000, C 0.000 }
gfCNCPoint4[8963] = {X 453.9149, Y 91.3787, Z -5.5000, A 0.000, B 0.000, C 0.000 }
gfCNCPoint4[8964] = {X 454.8963, Y 90.7176, Z -5.5000, A 0.000, B 0.000, C 0.000 }
gfCNCPoint4[8965] = {X 454.8963, Y 87.6139, Z -5.5000, A 0.000, B 0.000, C 0.000 }
gfCNCPoint4[8966] = {X 445.1937, Y 83.8105, Z -5.5000, A 0.000, B 0.000, C 0.000 }
gfCNCPoint4[8967] = {X 427.4646, Y 95.2951, Z -5.5000, A 0.000, B 0.000, C 0.000 }
gfCNCPoint4[8968] = {X 443.7032, Y 95.2951, Z -5.5000, A 0.000, B 0.000, C 0.000 }
gfCNCPoint4[8969] = {X 443.7032, Y 97.6951, Z -5.5000, A 0.000, B 0.000, C 0.000 }
gfCNCPoint4[8970] = {X 453.5796, Y 97.6951, Z -5.5000, A 0.000, B 0.000, C 0.000 }
gfCNCPoint4[8971] = {X 453.5796, Y 97.0659, Z -5.5000, A 0.000, B 0.000, C 0.000 }
gfCNCPoint4[8972] = {X 453.6990, Y 95.9930, Z -5.5000, A 0.000, B 0.000, C 0.000 }
gfCNCPoint4[8973] = {X 454.0514, Y 94.9725, Z -5.5000, A 0.000, B 0.000, C 0.000 }
gfCNCPoint4[8974] = {X 454.6196, Y 94.0545, Z -5.5000, A 0.000, B 0.000, C 0.000 }
gfCNCPoint4[8975] = {X 455.3757, Y 93.2839, Z -5.5000, A 0.000, B 0.000, C 0.000 }
gfCNCPoint4[8976] = {X 456.2827, Y 92.6984, Z -5.5000, A 0.000, B 0.000, C 0.000 }
gfCNCPoint4[8977] = {X 457.2963, Y 92.3266, Z -5.5000, A 0.000, B 0.000, C 0.000 }
gfCNCPoint4[8978] = {X 457.2963, Y 85.9769, Z -5.5000, A 0.000, B 0.000, C 0.000 }
gfCNCPoint4[8979] = {X 444.9227, Y 81.1265, Z -5.5000, A 0.000, B 0.000, C 0.000 }
gfCNCPoint4[8980] = {X 420.5856, Y 96.8916, Z -5.5000, A 0.000, B 0.000, C 0.000 }
gfCNCPoint4[8981] = {X 420.5867, Y 97.0659, Z -5.5000, A 0.000, B 0.000, C 0.000 }
gfCNCPoint4[8982] = {X 420.5867, Y 97.6951, Z -5.5000, A 0.000, B 0.000, C 0.000 }
gfCNCPoint4[8983] = {X 443.7032, Y 97.6951, Z -5.5000, A 0.000, B 0.000, C 0.000 }
gfCNCPoint4[8984] = {X 443.7032, Y 100.0951, Z -5.5000, A 0.000, B 0.000, C 0.000 }
gfCNCPoint4[8985] = {X 454.0522, Y 100.0951, Z -5.5000, A 0.000, B 0.000, C 0.000 }
gfCNCPoint4[8986] = {X 454.5210, Y 100.8812, Z -5.5000, A 0.000, B 0.000, C 0.000 }
gfCNCPoint4[8987] = {X 455.1283, Y 101.5661, Z -5.5000, A 0.000, B 0.000, C 0.000 }
gfCNCPoint4[8988] = {X 455.8528, Y 102.1254, Z -5.5000, A 0.000, B 0.000, C 0.000 }
gfCNCPoint4[8989] = {X 456.6691, Y 102.5396, Z -5.5000, A 0.000, B 0.000, C 0.000 }
gfCNCPoint4[8990] = {X 457.5483, Y 102.7942, Z -5.5000, A 0.000, B 0.000, C 0.000 }
gfCNCPoint4[8991] = {X 458.4596, Y 102.8800, Z -5.5000, A 0.000, B 0.000, C 0.000 }
gfCNCPoint4[8992] = {X 475.0000, Y 102.8800, Z -5.5000, A 0.000, B 0.000, C 0.000 }
gfCNCPoint4[8993] = {X 475.9113, Y 102.7942, Z -5.5000, A 0.000, B 0.000, C 0.000 }
gfCNCPoint4[8994] = {X 476.7905, Y 102.5396, Z -5.5000, A 0.000, B 0.000, C 0.000 }
gfCNCPoint4[8995] = {X 477.6068, Y 102.1254, Z -5.5000, A 0.000, B 0.000, C 0.000 }
gfCNCPoint4[8996] = {X 478.3313, Y 101.5661, Z -5.5000, A 0.000, B 0.000, C 0.000 }
gfCNCPoint4[8997] = {X 478.9386, Y 100.8812, Z -5.5000, A 0.000, B 0.000, C 0.000 }
gfCNCPoint4[8998] = {X 479.4074, Y 100.0951, Z -5.5000, A 0.000, B 0.000, C 0.000 }
gfCNCPoint4[8999] = {X 507.6814, Y 100.0951, Z -5.5000, A 0.000, B 0.000, C 0.000 }
gfCNCPoint4[9000] = {X 507.6814, Y 107.6951, Z -5.5000, A 0.000, B 0.000, C 0.000 }
gfCNCPoint4[9001] = {X 507.6814, Y 107.6951, Z -2.5000, A 0.000, B 0.000, C 0.000 }
gfCNCPoint4[9002] = {X 507.6814, Y 107.6951, Z 11.0000, A 0.000, B 0.000, C 0.000 }
gfCNCPoint4[9003] = {X 108.5565, Y 40.8987, Z 11.0000, A 0.000, B 0.000, C 0.000 }
gfCNCPoint4[9004] = {X 108.5565, Y 40.8987, Z -1.6667, A 0.000, B 0.000, C 0.000 }
gfCNCPoint4[9005] = {X 108.5565, Y 40.8987, Z -5.5000, A 0.000, B 0.000, C 0.000 }
gfCNCPoint4[9006] = {X 108.0674, Y 42.0939, Z -5.5000, A 0.000, B 0.000, C 0.000 }
gfCNCPoint4[9007] = {X 108.0973, Y 42.0419, Z -5.5000, A 0.000, B 0.000, C 0.000 }
gfCNCPoint4[9008] = {X 108.1278, Y 41.9904, Z -5.5000, A 0.000, B 0.000, C 0.000 }
gfCNCPoint4[9009] = {X 108.5501, Y 41.3806, Z -5.5000, A 0.000, B 0.000, C 0.000 }
gfCNCPoint4[9010] = {X 109.0456, Y 40.8286, Z -5.5000, A 0.000, B 0.000, C 0.000 }
gfCNCPoint4[9011] = {X 109.0455, Y 39.7036, Z -5.5000, A 0.000, B 0.000, C 0.000 }
gfCNCPoint4[9012] = {X 108.5565, Y 40.8987, Z -5.5000, A 0.000, B 0.000, C 0.000 }
gfCNCPoint4[9013] = {X 108.5565, Y 40.8987, Z -2.5000, A 0.000, B 0.000, C 0.000 }
gfCNCPoint4[9014] = {X 108.5565, Y 40.8987, Z 11.0000, A 0.000, B 0.000, C 0.000 }
gfCNCPoint4[9015] = {X 95.6829, Y 40.8728, Z 11.0000, A 0.000, B 0.000, C 0.000 }
gfCNCPoint4[9016] = {X 95.6829, Y 40.8728, Z -1.6667, A 0.000, B 0.000, C 0.000 }
gfCNCPoint4[9017] = {X 95.6829, Y 40.8728, Z -5.5000, A 0.000, B 0.000, C 0.000 }
gfCNCPoint4[9018] = {X 95.2114, Y 39.7196, Z -5.5000, A 0.000, B 0.000, C 0.000 }
gfCNCPoint4[9019] = {X 95.2114, Y 40.8685, Z -5.5000, A 0.000, B 0.000, C 0.000 }
gfCNCPoint4[9020] = {X 95.7315, Y 41.4077, Z -5.5000, A 0.000, B 0.000, C 0.000 }
gfCNCPoint4[9021] = {X 96.1544, Y 42.0260, Z -5.5000, A 0.000, B 0.000, C 0.000 }
gfCNCPoint4[9022] = {X 95.6829, Y 40.8728, Z -5.5000, A 0.000, B 0.000, C 0.000 }
gfCNCPoint4[9023] = {X 95.6829, Y 40.8728, Z -2.5000, A 0.000, B 0.000, C 0.000 }
gfCNCPoint4[9024] = {X 95.6829, Y 40.8728, Z 11.0000, A 0.000, B 0.000, C 0.000 }
gfCNCPoint4[9025] = {X -7.6966, Y 43.2914, Z 11.0000, A 0.000, B 0.000, C 0.000 }
gfCNCPoint4[9026] = {X -7.6966, Y 43.2914, Z -2.5000, A 0.000, B 0.000, C 0.000 }
gfCNCPoint4[9027] = {X -7.6966, Y 43.2914, Z -5.5000, A 0.000, B 0.000, C 0.000 }
gfCNCPoint4[9028] = {X -3.6966, Y 30.8006, Z -5.5000, A 0.000, B 0.000, C 0.000 }
gfCNCPoint4[9029] = {X -3.5208, Y 30.2844, Z -5.5000, A 0.000, B 0.000, C 0.000 }
gfCNCPoint4[9030] = {X -3.3262, Y 29.7750, Z -5.5000, A 0.000, B 0.000, C 0.000 }
gfCNCPoint4[9031] = {X -2.7032, Y 28.4548, Z -5.5000, A 0.000, B 0.000, C 0.000 }
gfCNCPoint4[9032] = {X -1.9094, Y 27.2298, Z -5.5000, A 0.000, B 0.000, C 0.000 }
gfCNCPoint4[9033] = {X -0.9591, Y 26.1217, Z -5.5000, A 0.000, B 0.000, C 0.000 }
gfCNCPoint4[9034] = {X 0.1306, Y 25.1505, Z -5.5000, A 0.000, B 0.000, C 0.000 }
gfCNCPoint4[9035] = {X 1.3404, Y 24.3336, Z -5.5000, A 0.000, B 0.000, C 0.000 }
gfCNCPoint4[9036] = {X 0.5799, Y 23.9234, Z -5.5000, A 0.000, B 0.000, C 0.000 }
gfCNCPoint4[9037] = {X -0.0858, Y 23.3724, Z -5.5000, A 0.000, B 0.000, C 0.000 }
gfCNCPoint4[9038] = {X -0.6309, Y 22.7019, Z -5.5000, A 0.000, B 0.000, C 0.000 }
gfCNCPoint4[9039] = {X -1.0345, Y 21.9378, Z -5.5000, A 0.000, B 0.000, C 0.000 }
gfCNCPoint4[9040] = {X -3.6458, Y 15.5423, Z -5.5000, A 0.000, B 0.000, C 0.000 }
gfCNCPoint4[9041] = {X -3.6717, Y 15.4773, Z -5.5000, A 0.000, B 0.000, C 0.000 }
gfCNCPoint4[9042] = {X -3.6966, Y 15.4119, Z -5.5000, A 0.000, B 0.000, C 0.000 }
gfCNCPoint4[9043] = {X -7.6966, Y 4.6488, Z -5.5000, A 0.000, B 0.000, C 0.000 }
gfCNCPoint4[9044] = {X -7.6966, Y 4.6488, Z -2.5000, A 0.000, B 0.000, C 0.000 }
gfCNCPoint4[9045] = {X -7.6966, Y 4.6488, Z 11.0000, A 0.000, B 0.000, C 0.000 }
gfCNCPoint4[9046] = {X -7.6966, Y 16.4128, Z 11.0000, A 0.000, B 0.000, C 0.000 }
gfCNCPoint4[9047] = {X -7.6966, Y 16.4128, Z -2.5000, A 0.000, B 0.000, C 0.000 }
gfCNCPoint4[9048] = {X -7.6966, Y 16.4128, Z -5.5000, A 0.000, B 0.000, C 0.000 }
gfCNCPoint4[9049] = {X -4.8866, Y 16.4128, Z -5.5000, A 0.000, B 0.000, C 0.000 }
gfCNCPoint4[9050] = {X -3.6966, Y 12.5939, Z -5.5000, A 0.000, B 0.000, C 0.000 }
gfCNCPoint4[9051] = {X -3.6606, Y 12.4835, Z -5.5000, A 0.000, B 0.000, C 0.000 }
gfCNCPoint4[9052] = {X -3.6216, Y 12.3742, Z -5.5000, A 0.000, B 0.000, C 0.000 }
gfCNCPoint4[9053] = {X -3.1667, Y 11.4828, Z -5.5000, A 0.000, B 0.000, C 0.000 }
gfCNCPoint4[9054] = {X -2.5189, Y 10.7201, Z -5.5000, A 0.000, B 0.000, C 0.000 }
gfCNCPoint4[9055] = {X -1.7129, Y 10.1268, Z -5.5000, A 0.000, B 0.000, C 0.000 }
gfCNCPoint4[9056] = {X -1.1157, Y 9.7861, Z -5.5000, A 0.000, B 0.000, C 0.000 }
gfCNCPoint4[9057] = {X -0.2303, Y 9.4048, Z -5.5000, A 0.000, B 0.000, C 0.000 }
gfCNCPoint4[9058] = {X 0.7176, Y 9.2294, Z -5.5000, A 0.000, B 0.000, C 0.000 }
gfCNCPoint4[9059] = {X 1.6808, Y 9.2686, Z -5.5000, A 0.000, B 0.000, C 0.000 }
gfCNCPoint4[9060] = {X 2.6114, Y 9.5203, Z -5.5000, A 0.000, B 0.000, C 0.000 }
gfCNCPoint4[9061] = {X 3.3911, Y 9.1469, Z -5.5000, A 0.000, B 0.000, C 0.000 }
gfCNCPoint4[9062] = {X 4.2001, Y 8.8419, Z -5.5000, A 0.000, B 0.000, C 0.000 }
gfCNCPoint4[9063] = {X 6.1105, Y 8.1738, Z -5.5000, A 0.000, B 0.000, C 0.000 }
gfCNCPoint4[9064] = {X 8.0713, Y 7.6728, Z -5.5000, A 0.000, B 0.000, C 0.000 }
gfCNCPoint4[9065] = {X 10.0681, Y 7.3426, Z -5.5000, A 0.000, B 0.000, C 0.000 }
gfCNCPoint4[9066] = {X 12.0859, Y 7.1857, Z -5.5000, A 0.000, B 0.000, C 0.000 }
gfCNCPoint4[9067] = {X 14.1097, Y 7.2032, Z -5.5000, A 0.000, B 0.000, C 0.000 }
gfCNCPoint4[9068] = {X 16.1244, Y 7.3951, Z -5.5000, A 0.000, B 0.000, C 0.000 }
gfCNCPoint4[9069] = {X 17.9477, Y 7.7286, Z -5.5000, A 0.000, B 0.000, C 0.000 }
gfCNCPoint4[9070] = {X 19.7252, Y 8.2536, Z -5.5000, A 0.000, B 0.000, C 0.000 }
gfCNCPoint4[9071] = {X 21.4371, Y 8.9642, Z -5.5000, A 0.000, B 0.000, C 0.000 }
gfCNCPoint4[9072] = {X 23.0639, Y 9.8523, Z -5.5000, A 0.000, B 0.000, C 0.000 }
gfCNCPoint4[9073] = {X 24.5874, Y 10.9080, Z -5.5000, A 0.000, B 0.000, C 0.000 }
gfCNCPoint4[9074] = {X 25.6727, Y 11.8569, Z -5.5000, A 0.000, B 0.000, C 0.000 }
gfCNCPoint4[9075] = {X 26.6463, Y 12.9202, Z -5.5000, A 0.000, B 0.000, C 0.000 }
gfCNCPoint4[9076] = {X 27.4962, Y 14.0848, Z -5.5000, A 0.000, B 0.000, C 0.000 }
gfCNCPoint4[9077] = {X 28.2118, Y 15.3363, Z -5.5000, A 0.000, B 0.000, C 0.000 }
gfCNCPoint4[9078] = {X 28.7845, Y 16.6593, Z -5.5000, A 0.000, B 0.000, C 0.000 }
gfCNCPoint4[9079] = {X 29.2595, Y 18.3155, Z -5.5000, A 0.000, B 0.000, C 0.000 }
gfCNCPoint4[9080] = {X 29.5414, Y 20.0152, Z -5.5000, A 0.000, B 0.000, C 0.000 }
gfCNCPoint4[9081] = {X 29.6265, Y 21.7360, Z -5.5000, A 0.000, B 0.000, C 0.000 }
gfCNCPoint4[9082] = {X 29.5136, Y 23.4553, Z -5.5000, A 0.000, B 0.000, C 0.000 }
gfCNCPoint4[9083] = {X 29.2042, Y 25.1502, Z -5.5000, A 0.000, B 0.000, C 0.000 }
gfCNCPoint4[9084] = {X 28.7619, Y 26.5966, Z -5.5000, A 0.000, B 0.000, C 0.000 }
gfCNCPoint4[9085] = {X 28.1366, Y 27.9738, Z -5.5000, A 0.000, B 0.000, C 0.000 }
gfCNCPoint4[9086] = {X 27.3388, Y 29.2587, Z -5.5000, A 0.000, B 0.000, C 0.000 }
gfCNCPoint4[9087] = {X 26.3818, Y 30.4299, Z -5.5000, A 0.000, B 0.000, C 0.000 }
gfCNCPoint4[9088] = {X 25.2815, Y 31.4678, Z -5.5000, A 0.000, B 0.000, C 0.000 }
gfCNCPoint4[9089] = {X 26.0854, Y 31.8099, Z -5.5000, A 0.000, B 0.000, C 0.000 }
gfCNCPoint4[9090] = {X 26.8041, Y 32.3068, Z -5.5000, A 0.000, B 0.000, C 0.000 }
gfCNCPoint4[9091] = {X 27.4080, Y 32.9382, Z -5.5000, A 0.000, B 0.000, C 0.000 }
gfCNCPoint4[9092] = {X 27.8726, Y 33.6781, Z -5.5000, A 0.000, B 0.000, C 0.000 }
gfCNCPoint4[9093] = {X 30.9100, Y 39.9530, Z -5.5000, A 0.000, B 0.000, C 0.000 }
gfCNCPoint4[9094] = {X 31.2306, Y 40.8622, Z -5.5000, A 0.000, B 0.000, C 0.000 }
gfCNCPoint4[9095] = {X 31.3415, Y 41.8197, Z -5.5000, A 0.000, B 0.000, C 0.000 }
gfCNCPoint4[9096] = {X 31.2374, Y 42.7781, Z -5.5000, A 0.000, B 0.000, C 0.000 }
gfCNCPoint4[9097] = {X 30.9234, Y 43.6895, Z -5.5000, A 0.000, B 0.000, C 0.000 }
gfCNCPoint4[9098] = {X 30.4150, Y 44.5085, Z -5.5000, A 0.000, B 0.000, C 0.000 }
gfCNCPoint4[9099] = {X 29.7377, Y 45.1945, Z -5.5000, A 0.000, B 0.000, C 0.000 }
gfCNCPoint4[9100] = {X 29.2016, Y 45.6279, Z -5.5000, A 0.000, B 0.000, C 0.000 }
gfCNCPoint4[9101] = {X 28.4975, Y 46.0915, Z -5.5000, A 0.000, B 0.000, C 0.000 }
gfCNCPoint4[9102] = {X 27.7170, Y 46.4099, Z -5.5000, A 0.000, B 0.000, C 0.000 }
gfCNCPoint4[9103] = {X 26.8896, Y 46.5712, Z -5.5000, A 0.000, B 0.000, C 0.000 }
gfCNCPoint4[9104] = {X 26.0467, Y 46.5692, Z -5.5000, A 0.000, B 0.000, C 0.000 }
gfCNCPoint4[9105] = {X 25.2201, Y 46.4040, Z -5.5000, A 0.000, B 0.000, C 0.000 }
gfCNCPoint4[9106] = {X 23.4200, Y 47.3543, Z -5.5000, A 0.000, B 0.000, C 0.000 }
gfCNCPoint4[9107] = {X 21.5581, Y 48.1769, Z -5.5000, A 0.000, B 0.000, C 0.000 }
gfCNCPoint4[9108] = {X 19.6434, Y 48.8677, Z -5.5000, A 0.000, B 0.000, C 0.000 }
gfCNCPoint4[9109] = {X 17.7035, Y 49.4150, Z -5.5000, A 0.000, B 0.000, C 0.000 }
gfCNCPoint4[9110] = {X 15.7229, Y 49.7886, Z -5.5000, A 0.000, B 0.000, C 0.000 }
gfCNCPoint4[9111] = {X 13.7170, Y 49.9856, Z -5.5000, A 0.000, B 0.000, C 0.000 }
gfCNCPoint4[9112] = {X 11.7015, Y 50.0043, Z -5.5000, A 0.000, B 0.000, C 0.000 }
gfCNCPoint4[9113] = {X 9.6922, Y 49.8447, Z -5.5000, A 0.000, B 0.000, C 0.000 }
gfCNCPoint4[9114] = {X 7.7050, Y 49.5080, Z -5.5000, A 0.000, B 0.000, C 0.000 }
gfCNCPoint4[9115] = {X 5.8034, Y 48.9874, Z -5.5000, A 0.000, B 0.000, C 0.000 }
gfCNCPoint4[9116] = {X 3.9766, Y 48.2463, Z -5.5000, A 0.000, B 0.000, C 0.000 }
gfCNCPoint4[9117] = {X 2.2498, Y 47.2949, Z -5.5000, A 0.000, B 0.000, C 0.000 }
gfCNCPoint4[9118] = {X 0.6472, Y 46.1466, Z -5.5000, A 0.000, B 0.000, C 0.000 }
gfCNCPoint4[9119] = {X -0.4853, Y 45.1287, Z -5.5000, A 0.000, B 0.000, C 0.000 }
gfCNCPoint4[9120] = {X -1.4912, Y 43.9854, Z -5.5000, A 0.000, B 0.000, C 0.000 }
gfCNCPoint4[9121] = {X -2.3565, Y 42.7324, Z -5.5000, A 0.000, B 0.000, C 0.000 }
gfCNCPoint4[9122] = {X -3.0695, Y 41.3869, Z -5.5000, A 0.000, B 0.000, C 0.000 }
gfCNCPoint4[9123] = {X -3.6205, Y 39.9673, Z -5.5000, A 0.000, B 0.000, C 0.000 }
gfCNCPoint4[9124] = {X -3.6591, Y 39.8451, Z -5.5000, A 0.000, B 0.000, C 0.000 }
gfCNCPoint4[9125] = {X -3.6966, Y 39.7227, Z -5.5000, A 0.000, B 0.000, C 0.000 }
gfCNCPoint4[9126] = {X -4.8478, Y 35.8919, Z -5.5000, A 0.000, B 0.000, C 0.000 }
gfCNCPoint4[9127] = {X -7.9945, Y 36.0044, Z -5.5000, A 0.000, B 0.000, C 0.000 }
gfCNCPoint4[9128] = {X -7.9945, Y 36.0044, Z -2.5000, A 0.000, B 0.000, C 0.000 }
gfCNCPoint4[9129] = {X -7.9945, Y 36.0044, Z 11.0000, A 0.000, B 0.000, C 0.000 }
gfCNCPoint4[9130] = {X 608.0000, Y 40.1195, Z 11.0000, A 0.000, B 0.000, C 0.000 }
gfCNCPoint4[9131] = {X 608.0000, Y 40.1195, Z -2.5000, A 0.000, B 0.000, C 0.000 }
gfCNCPoint4[9132] = {X 608.0000, Y 40.1195, Z -5.5000, A 0.000, B 0.000, C 0.000 }
gfCNCPoint4[9133] = {X 603.6966, Y 47.2355, Z -5.5000, A 0.000, B 0.000, C 0.000 }
gfCNCPoint4[9134] = {X 603.6634, Y 47.2895, Z -5.5000, A 0.000, B 0.000, C 0.000 }
gfCNCPoint4[9135] = {X 603.6294, Y 47.3431, Z -5.5000, A 0.000, B 0.000, C 0.000 }
gfCNCPoint4[9136] = {X 603.0930, Y 48.0159, Z -5.5000, A 0.000, B 0.000, C 0.000 }
gfCNCPoint4[9137] = {X 602.4340, Y 48.5690, Z -5.5000, A 0.000, B 0.000, C 0.000 }
gfCNCPoint4[9138] = {X 601.6784, Y 48.9806, Z -5.5000, A 0.000, B 0.000, C 0.000 }
gfCNCPoint4[9139] = {X 600.8562, Y 49.2343, Z -5.5000, A 0.000, B 0.000, C 0.000 }
gfCNCPoint4[9140] = {X 600.0000, Y 49.3200, Z -5.5000, A 0.000, B 0.000, C 0.000 }
gfCNCPoint4[9141] = {X 593.5565, Y 49.3200, Z -5.5000, A 0.000, B 0.000, C 0.000 }
gfCNCPoint4[9142] = {X 592.5952, Y 49.2117, Z -5.5000, A 0.000, B 0.000, C 0.000 }
gfCNCPoint4[9143] = {X 591.6822, Y 48.8922, Z -5.5000, A 0.000, B 0.000, C 0.000 }
gfCNCPoint4[9144] = {X 590.8631, Y 48.3775, Z -5.5000, A 0.000, B 0.000, C 0.000 }
gfCNCPoint4[9145] = {X 590.1790, Y 47.6935, Z -5.5000, A 0.000, B 0.000, C 0.000 }
gfCNCPoint4[9146] = {X 589.6643, Y 46.8744, Z -5.5000, A 0.000, B 0.000, C 0.000 }
gfCNCPoint4[9147] = {X 589.3448, Y 45.9613, Z -5.5000, A 0.000, B 0.000, C 0.000 }
gfCNCPoint4[9148] = {X 589.2365, Y 45.0000, Z -5.5000, A 0.000, B 0.000, C 0.000 }
gfCNCPoint4[9149] = {X 589.2365, Y 44.0646, Z -5.5000, A 0.000, B 0.000, C 0.000 }
gfCNCPoint4[9150] = {X 589.3406, Y 43.1363, Z -5.5000, A 0.000, B 0.000, C 0.000 }
gfCNCPoint4[9151] = {X 589.6401, Y 42.2515, Z -5.5000, A 0.000, B 0.000, C 0.000 }
gfCNCPoint4[9152] = {X 590.1212, Y 41.4508, Z -5.5000, A 0.000, B 0.000, C 0.000 }
gfCNCPoint4[9153] = {X 590.7619, Y 40.7710, Z -5.5000, A 0.000, B 0.000, C 0.000 }
gfCNCPoint4[9154] = {X 590.7625, Y 33.5316, Z -5.5000, A 0.000, B 0.000, C 0.000 }
gfCNCPoint4[9155] = {X 585.4453, Y 46.6524, Z -5.5000, A 0.000, B 0.000, C 0.000 }
gfCNCPoint4[9156] = {X 585.0755, Y 47.3550, Z -5.5000, A 0.000, B 0.000, C 0.000 }
gfCNCPoint4[9157] = {X 584.5834, Y 47.9780, Z -5.5000, A 0.000, B 0.000, C 0.000 }
gfCNCPoint4[9158] = {X 583.9856, Y 48.5004, Z -5.5000, A 0.000, B 0.000, C 0.000 }
gfCNCPoint4[9159] = {X 583.3023, Y 48.9046, Z -5.5000, A 0.000, B 0.000, C 0.000 }
gfCNCPoint4[9160] = {X 582.3585, Y 49.2242, Z -5.5000, A 0.000, B 0.000, C 0.000 }
gfCNCPoint4[9161] = {X 581.3666, Y 49.3191, Z -5.5000, A 0.000, B 0.000, C 0.000 }
gfCNCPoint4[9162] = {X 580.3794, Y 49.1842, Z -5.5000, A 0.000, B 0.000, C 0.000 }
gfCNCPoint4[9163] = {X 579.4493, Y 48.8268, Z -5.5000, A 0.000, B 0.000, C 0.000 }
gfCNCPoint4[9164] = {X 578.6259, Y 48.2657, Z -5.5000, A 0.000, B 0.000, C 0.000 }
gfCNCPoint4[9165] = {X 577.9529, Y 47.5309, Z -5.5000, A 0.000, B 0.000, C 0.000 }
gfCNCPoint4[9166] = {X 577.4662, Y 46.6615, Z -5.5000, A 0.000, B 0.000, C 0.000 }
gfCNCPoint4[9167] = {X 572.0192, Y 33.3423, Z -5.5000, A 0.000, B 0.000, C 0.000 }
gfCNCPoint4[9168] = {X 572.0222, Y 40.7726, Z -5.5000, A 0.000, B 0.000, C 0.000 }
gfCNCPoint4[9169] = {X 572.6594, Y 41.4435, Z -5.5000, A 0.000, B 0.000, C 0.000 }
gfCNCPoint4[9170] = {X 573.1391, Y 42.2346, Z -5.5000, A 0.000, B 0.000, C 0.000 }
gfCNCPoint4[9171] = {X 573.4393, Y 43.1097, Z -5.5000, A 0.000, B 0.000, C 0.000 }
gfCNCPoint4[9172] = {X 573.5463, Y 44.0287, Z -5.5000, A 0.000, B 0.000, C 0.000 }
gfCNCPoint4[9173] = {X 573.5464, Y 45.0000, Z -5.5000, A 0.000, B 0.000, C 0.000 }
gfCNCPoint4[9174] = {X 573.4381, Y 45.9613, Z -5.5000, A 0.000, B 0.000, C 0.000 }
gfCNCPoint4[9175] = {X 573.1186, Y 46.8744, Z -5.5000, A 0.000, B 0.000, C 0.000 }
gfCNCPoint4[9176] = {X 572.6039, Y 47.6935, Z -5.5000, A 0.000, B 0.000, C 0.000 }
gfCNCPoint4[9177] = {X 571.9199, Y 48.3775, Z -5.5000, A 0.000, B 0.000, C 0.000 }
gfCNCPoint4[9178] = {X 571.1008, Y 48.8922, Z -5.5000, A 0.000, B 0.000, C 0.000 }
gfCNCPoint4[9179] = {X 570.1877, Y 49.2117, Z -5.5000, A 0.000, B 0.000, C 0.000 }
gfCNCPoint4[9180] = {X 569.2264, Y 49.3200, Z -5.5000, A 0.000, B 0.000, C 0.000 }
gfCNCPoint4[9181] = {X 562.4443, Y 49.3200, Z -5.5000, A 0.000, B 0.000, C 0.000 }
gfCNCPoint4[9182] = {X 561.4830, Y 49.2117, Z -5.5000, A 0.000, B 0.000, C 0.000 }
gfCNCPoint4[9183] = {X 560.5699, Y 48.8922, Z -5.5000, A 0.000, B 0.000, C 0.000 }
gfCNCPoint4[9184] = {X 559.7508, Y 48.3775, Z -5.5000, A 0.000, B 0.000, C 0.000 }
gfCNCPoint4[9185] = {X 559.0668, Y 47.6935, Z -5.5000, A 0.000, B 0.000, C 0.000 }
gfCNCPoint4[9186] = {X 558.5521, Y 46.8744, Z -5.5000, A 0.000, B 0.000, C 0.000 }
gfCNCPoint4[9187] = {X 558.2326, Y 45.9613, Z -5.5000, A 0.000, B 0.000, C 0.000 }
gfCNCPoint4[9188] = {X 558.1243, Y 45.0000, Z -5.5000, A 0.000, B 0.000, C 0.000 }
gfCNCPoint4[9189] = {X 558.1243, Y 44.0647, Z -5.5000, A 0.000, B 0.000, C 0.000 }
gfCNCPoint4[9190] = {X 558.2282, Y 43.1360, Z -5.5000, A 0.000, B 0.000, C 0.000 }
gfCNCPoint4[9191] = {X 558.5280, Y 42.2509, Z -5.5000, A 0.000, B 0.000, C 0.000 }
gfCNCPoint4[9192] = {X 559.0098, Y 41.4502, Z -5.5000, A 0.000, B 0.000, C 0.000 }
gfCNCPoint4[9193] = {X 559.6515, Y 40.7707, Z -5.5000, A 0.000, B 0.000, C 0.000 }
gfCNCPoint4[9194] = {X 559.6515, Y 9.2299, Z -5.5000, A 0.000, B 0.000, C 0.000 }
gfCNCPoint4[9195] = {X 559.0132, Y 8.5590, Z -5.5000, A 0.000, B 0.000, C 0.000 }
gfCNCPoint4[9196] = {X 558.5326, Y 7.7674, Z -5.5000, A 0.000, B 0.000, C 0.000 }
gfCNCPoint4[9197] = {X 558.2318, Y 6.8916, Z -5.5000, A 0.000, B 0.000, C 0.000 }
gfCNCPoint4[9198] = {X 558.1245, Y 5.9718, Z -5.5000, A 0.000, B 0.000, C 0.000 }
gfCNCPoint4[9199] = {X 558.1243, Y 5.0000, Z -5.5000, A 0.000, B 0.000, C 0.000 }
gfCNCPoint4[9200] = {X 558.2326, Y 4.0387, Z -5.5000, A 0.000, B 0.000, C 0.000 }
gfCNCPoint4[9201] = {X 558.5521, Y 3.1256, Z -5.5000, A 0.000, B 0.000, C 0.000 }
gfCNCPoint4[9202] = {X 559.0668, Y 2.3065, Z -5.5000, A 0.000, B 0.000, C 0.000 }
gfCNCPoint4[9203] = {X 559.7508, Y 1.6225, Z -5.5000, A 0.000, B 0.000, C 0.000 }
gfCNCPoint4[9204] = {X 560.5699, Y 1.1078, Z -5.5000, A 0.000, B 0.000, C 0.000 }
gfCNCPoint4[9205] = {X 561.4830, Y 0.7883, Z -5.5000, A 0.000, B 0.000, C 0.000 }
gfCNCPoint4[9206] = {X 562.4443, Y 0.6800, Z -5.5000, A 0.000, B 0.000, C 0.000 }
gfCNCPoint4[9207] = {X 570.9376, Y 0.6800, Z -5.5000, A 0.000, B 0.000, C 0.000 }
gfCNCPoint4[9208] = {X 571.8988, Y 0.7883, Z -5.5000, A 0.000, B 0.000, C 0.000 }
gfCNCPoint4[9209] = {X 572.8119, Y 1.1078, Z -5.5000, A 0.000, B 0.000, C 0.000 }
gfCNCPoint4[9210] = {X 573.6310, Y 1.6225, Z -5.5000, A 0.000, B 0.000, C 0.000 }
gfCNCPoint4[9211] = {X 574.3151, Y 2.3065, Z -5.5000, A 0.000, B 0.000, C 0.000 }
gfCNCPoint4[9212] = {X 574.8297, Y 3.1256, Z -5.5000, A 0.000, B 0.000, C 0.000 }
gfCNCPoint4[9213] = {X 575.1492, Y 4.0387, Z -5.5000, A 0.000, B 0.000, C 0.000 }
gfCNCPoint4[9214] = {X 575.2576, Y 5.0000, Z -5.5000, A 0.000, B 0.000, C 0.000 }
gfCNCPoint4[9215] = {X 575.2576, Y 5.9342, Z -5.5000, A 0.000, B 0.000, C 0.000 }
gfCNCPoint4[9216] = {X 575.1835, Y 6.7304, Z -5.5000, A 0.000, B 0.000, C 0.000 }
gfCNCPoint4[9217] = {X 574.9640, Y 7.4993, Z -5.5000, A 0.000, B 0.000, C 0.000 }
gfCNCPoint4[9218] = {X 574.6066, Y 8.2146, Z -5.5000, A 0.000, B 0.000, C 0.000 }
gfCNCPoint4[9219] = {X 581.1910, Y 24.3695, Z -5.5000, A 0.000, B 0.000, C 0.000 }
gfCNCPoint4[9220] = {X 587.8457, Y 8.0940, Z -5.5000, A 0.000, B 0.000, C 0.000 }
gfCNCPoint4[9221] = {X 587.5316, Y 7.4229, Z -5.5000, A 0.000, B 0.000, C 0.000 }
gfCNCPoint4[9222] = {X 587.3369, Y 6.7081, Z -5.5000, A 0.000, B 0.000, C 0.000 }
gfCNCPoint4[9223] = {X 587.2671, Y 5.9705, Z -5.5000, A 0.000, B 0.000, C 0.000 }
gfCNCPoint4[9224] = {X 587.2670, Y 5.0000, Z -5.5000, A 0.000, B 0.000, C 0.000 }
gfCNCPoint4[9225] = {X 587.3753, Y 4.0387, Z -5.5000, A 0.000, B 0.000, C 0.000 }
gfCNCPoint4[9226] = {X 587.6948, Y 3.1256, Z -5.5000, A 0.000, B 0.000, C 0.000 }
gfCNCPoint4[9227] = {X 588.2094, Y 2.3065, Z -5.5000, A 0.000, B 0.000, C 0.000 }
gfCNCPoint4[9228] = {X 588.8935, Y 1.6225, Z -5.5000, A 0.000, B 0.000, C 0.000 }
gfCNCPoint4[9229] = {X 589.7126, Y 1.1078, Z -5.5000, A 0.000, B 0.000, C 0.000 }
gfCNCPoint4[9230] = {X 590.6257, Y 0.7883, Z -5.5000, A 0.000, B 0.000, C 0.000 }
gfCNCPoint4[9231] = {X 591.5870, Y 0.6800, Z -5.5000, A 0.000, B 0.000, C 0.000 }
gfCNCPoint4[9232] = {X 600.0000, Y 0.6800, Z -5.5000, A 0.000, B 0.000, C 0.000 }
gfCNCPoint4[9233] = {X 600.8562, Y 0.7657, Z -5.5000, A 0.000, B 0.000, C 0.000 }
gfCNCPoint4[9234] = {X 601.6784, Y 1.0194, Z -5.5000, A 0.000, B 0.000, C 0.000 }
gfCNCPoint4[9235] = {X 602.4340, Y 1.4310, Z -5.5000, A 0.000, B 0.000, C 0.000 }
gfCNCPoint4[9236] = {X 603.0930, Y 1.9841, Z -5.5000, A 0.000, B 0.000, C 0.000 }
gfCNCPoint4[9237] = {X 603.6294, Y 2.6569, Z -5.5000, A 0.000, B 0.000, C 0.000 }
gfCNCPoint4[9238] = {X 603.6634, Y 2.7105, Z -5.5000, A 0.000, B 0.000, C 0.000 }
gfCNCPoint4[9239] = {X 603.6966, Y 2.7645, Z -5.5000, A 0.000, B 0.000, C 0.000 }
gfCNCPoint4[9240] = {X 608.0000, Y 9.8805, Z -5.5000, A 0.000, B 0.000, C 0.000 }
gfCNCPoint4[9241] = {X 608.0000, Y 9.8805, Z -2.5000, A 0.000, B 0.000, C 0.000 }
gfCNCPoint4[9242] = {X 608.0000, Y 9.8805, Z 11.0000, A 0.000, B 0.000, C 0.000 }
gfCNCPoint4[9243] = {X -7.6966, Y 16.7867, Z 11.0000, A 0.000, B 0.000, C 0.000 }
gfCNCPoint4[9244] = {X -7.6966, Y 16.7867, Z -2.5000, A 0.000, B 0.000, C 0.000 }
gfCNCPoint4[9245] = {X -7.6966, Y 16.7867, Z -5.5000, A 0.000, B 0.000, C 0.000 }
gfCNCPoint4[9246] = {X -4.6243, Y 16.7867, Z -5.5000, A 0.000, B 0.000, C 0.000 }
gfCNCPoint4[9247] = {X -3.6966, Y 12.8957, Z -5.5000, A 0.000, B 0.000, C 0.000 }
gfCNCPoint4[9248] = {X -3.6291, Y 12.6466, Z -5.5000, A 0.000, B 0.000, C 0.000 }
gfCNCPoint4[9249] = {X -3.5466, Y 12.4021, Z -5.5000, A 0.000, B 0.000, C 0.000 }
gfCNCPoint4[9250] = {X -3.1001, Y 11.5272, Z -5.5000, A 0.000, B 0.000, C 0.000 }
gfCNCPoint4[9251] = {X -2.4643, Y 10.7786, Z -5.5000, A 0.000, B 0.000, C 0.000 }
gfCNCPoint4[9252] = {X -1.6733, Y 10.1963, Z -5.5000, A 0.000, B 0.000, C 0.000 }
gfCNCPoint4[9253] = {X -1.0760, Y 9.8556, Z -5.5000, A 0.000, B 0.000, C 0.000 }
gfCNCPoint4[9254] = {X -0.1982, Y 9.4787, Z -5.5000, A 0.000, B 0.000, C 0.000 }
gfCNCPoint4[9255] = {X 0.7417, Y 9.3079, Z -5.5000, A 0.000, B 0.000, C 0.000 }
gfCNCPoint4[9256] = {X 1.6960, Y 9.3519, Z -5.5000, A 0.000, B 0.000, C 0.000 }
gfCNCPoint4[9257] = {X 2.6163, Y 9.6084, Z -5.5000, A 0.000, B 0.000, C 0.000 }
gfCNCPoint4[9258] = {X 3.4066, Y 9.2272, Z -5.5000, A 0.000, B 0.000, C 0.000 }
gfCNCPoint4[9259] = {X 4.2274, Y 8.9171, Z -5.5000, A 0.000, B 0.000, C 0.000 }
gfCNCPoint4[9260] = {X 6.1317, Y 8.2509, Z -5.5000, A 0.000, B 0.000, C 0.000 }
gfCNCPoint4[9261] = {X 8.0863, Y 7.7514, Z -5.5000, A 0.000, B 0.000, C 0.000 }
gfCNCPoint4[9262] = {X 10.0767, Y 7.4221, Z -5.5000, A 0.000, B 0.000, C 0.000 }
gfCNCPoint4[9263] = {X 12.0881, Y 7.2656, Z -5.5000, A 0.000, B 0.000, C 0.000 }
gfCNCPoint4[9264] = {X 14.1054, Y 7.2831, Z -5.5000, A 0.000, B 0.000, C 0.000 }
gfCNCPoint4[9265] = {X 16.1138, Y 7.4744, Z -5.5000, A 0.000, B 0.000, C 0.000 }
gfCNCPoint4[9266] = {X 17.9288, Y 7.8064, Z -5.5000, A 0.000, B 0.000, C 0.000 }
gfCNCPoint4[9267] = {X 19.6983, Y 8.3289, Z -5.5000, A 0.000, B 0.000, C 0.000 }
gfCNCPoint4[9268] = {X 21.4024, Y 9.0363, Z -5.5000, A 0.000, B 0.000, C 0.000 }
gfCNCPoint4[9269] = {X 23.0218, Y 9.9204, Z -5.5000, A 0.000, B 0.000, C 0.000 }
gfCNCPoint4[9270] = {X 24.5384, Y 10.9713, Z -5.5000, A 0.000, B 0.000, C 0.000 }
gfCNCPoint4[9271] = {X 25.6170, Y 11.9143, Z -5.5000, A 0.000, B 0.000, C 0.000 }
gfCNCPoint4[9272] = {X 26.5845, Y 12.9710, Z -5.5000, A 0.000, B 0.000, C 0.000 }
gfCNCPoint4[9273] = {X 27.4291, Y 14.1284, Z -5.5000, A 0.000, B 0.000, C 0.000 }
gfCNCPoint4[9274] = {X 28.1403, Y 15.3721, Z -5.5000, A 0.000, B 0.000, C 0.000 }
gfCNCPoint4[9275] = {X 28.7095, Y 16.6870, Z -5.5000, A 0.000, B 0.000, C 0.000 }
gfCNCPoint4[9276] = {X 29.1818, Y 18.3341, Z -5.5000, A 0.000, B 0.000, C 0.000 }
gfCNCPoint4[9277] = {X 29.4620, Y 20.0246, Z -5.5000, A 0.000, B 0.000, C 0.000 }
gfCNCPoint4[9278] = {X 29.5465, Y 21.7360, Z -5.5000, A 0.000, B 0.000, C 0.000 }
gfCNCPoint4[9279] = {X 29.4341, Y 23.4459, Z -5.5000, A 0.000, B 0.000, C 0.000 }
gfCNCPoint4[9280] = {X 29.1264, Y 25.1315, Z -5.5000, A 0.000, B 0.000, C 0.000 }
gfCNCPoint4[9281] = {X 28.6764, Y 26.5964, Z -5.5000, A 0.000, B 0.000, C 0.000 }
gfCNCPoint4[9282] = {X 28.0374, Y 27.9893, Z -5.5000, A 0.000, B 0.000, C 0.000 }
gfCNCPoint4[9283] = {X 27.2206, Y 29.2859, Z -5.5000, A 0.000, B 0.000, C 0.000 }
gfCNCPoint4[9284] = {X 26.2401, Y 30.4637, Z -5.5000, A 0.000, B 0.000, C 0.000 }
gfCNCPoint4[9285] = {X 25.1131, Y 31.5020, Z -5.5000, A 0.000, B 0.000, C 0.000 }
gfCNCPoint4[9286] = {X 25.2526, Y 31.5426, Z -5.5000, A 0.000, B 0.000, C 0.000 }
gfCNCPoint4[9287] = {X 25.3907, Y 31.5878, Z -5.5000, A 0.000, B 0.000, C 0.000 }
gfCNCPoint4[9288] = {X 26.1381, Y 31.9317, Z -5.5000, A 0.000, B 0.000, C 0.000 }
gfCNCPoint4[9289] = {X 26.8050, Y 32.4135, Z -5.5000, A 0.000, B 0.000, C 0.000 }
gfCNCPoint4[9290] = {X 27.3663, Y 33.0150, Z -5.5000, A 0.000, B 0.000, C 0.000 }
gfCNCPoint4[9291] = {X 27.8009, Y 33.7136, Z -5.5000, A 0.000, B 0.000, C 0.000 }
gfCNCPoint4[9292] = {X 30.8380, Y 39.9879, Z -5.5000, A 0.000, B 0.000, C 0.000 }
gfCNCPoint4[9293] = {X 31.1526, Y 40.8802, Z -5.5000, A 0.000, B 0.000, C 0.000 }
gfCNCPoint4[9294] = {X 31.2615, Y 41.8200, Z -5.5000, A 0.000, B 0.000, C 0.000 }
gfCNCPoint4[9295] = {X 31.1593, Y 42.7606, Z -5.5000, A 0.000, B 0.000, C 0.000 }
gfCNCPoint4[9296] = {X 30.8511, Y 43.6551, Z -5.5000, A 0.000, B 0.000, C 0.000 }
gfCNCPoint4[9297] = {X 30.3522, Y 44.4590, Z -5.5000, A 0.000, B 0.000, C 0.000 }
gfCNCPoint4[9298] = {X 29.6874, Y 45.1323, Z -5.5000, A 0.000, B 0.000, C 0.000 }
gfCNCPoint4[9299] = {X 29.1513, Y 45.5657, Z -5.5000, A 0.000, B 0.000, C 0.000 }
gfCNCPoint4[9300] = {X 28.4542, Y 46.0239, Z -5.5000, A 0.000, B 0.000, C 0.000 }
gfCNCPoint4[9301] = {X 27.6810, Y 46.3372, Z -5.5000, A 0.000, B 0.000, C 0.000 }
gfCNCPoint4[9302] = {X 26.8615, Y 46.4935, Z -5.5000, A 0.000, B 0.000, C 0.000 }
gfCNCPoint4[9303] = {X 26.0272, Y 46.4868, Z -5.5000, A 0.000, B 0.000, C 0.000 }
gfCNCPoint4[9304] = {X 25.2104, Y 46.3173, Z -5.5000, A 0.000, B 0.000, C 0.000 }
gfCNCPoint4[9305] = {X 23.4059, Y 47.2723, Z -5.5000, A 0.000, B 0.000, C 0.000 }
gfCNCPoint4[9306] = {X 21.5389, Y 48.0984, Z -5.5000, A 0.000, B 0.000, C 0.000 }
gfCNCPoint4[9307] = {X 19.6185, Y 48.7916, Z -5.5000, A 0.000, B 0.000, C 0.000 }
gfCNCPoint4[9308] = {X 17.6855, Y 49.3371, Z -5.5000, A 0.000, B 0.000, C 0.000 }
gfCNCPoint4[9309] = {X 15.7117, Y 49.7094, Z -5.5000, A 0.000, B 0.000, C 0.000 }
gfCNCPoint4[9310] = {X 13.7128, Y 49.9057, Z -5.5000, A 0.000, B 0.000, C 0.000 }
gfCNCPoint4[9311] = {X 11.7043, Y 49.9244, Z -5.5000, A 0.000, B 0.000, C 0.000 }
gfCNCPoint4[9312] = {X 9.7020, Y 49.7653, Z -5.5000, A 0.000, B 0.000, C 0.000 }
gfCNCPoint4[9313] = {X 7.7217, Y 49.4297, Z -5.5000, A 0.000, B 0.000, C 0.000 }
gfCNCPoint4[9314] = {X 5.8292, Y 48.9116, Z -5.5000, A 0.000, B 0.000, C 0.000 }
gfCNCPoint4[9315] = {X 4.0109, Y 48.1740, Z -5.5000, A 0.000, B 0.000, C 0.000 }
gfCNCPoint4[9316] = {X 2.2923, Y 47.2272, Z -5.5000, A 0.000, B 0.000, C 0.000 }
gfCNCPoint4[9317] = {X 0.6974, Y 46.0843, Z -5.5000, A 0.000, B 0.000, C 0.000 }
gfCNCPoint4[9318] = {X -0.4283, Y 45.0726, Z -5.5000, A 0.000, B 0.000, C 0.000 }
gfCNCPoint4[9319] = {X -1.4280, Y 43.9363, Z -5.5000, A 0.000, B 0.000, C 0.000 }
gfCNCPoint4[9320] = {X -2.2881, Y 42.6910, Z -5.5000, A 0.000, B 0.000, C 0.000 }
gfCNCPoint4[9321] = {X -2.9968, Y 41.3537, Z -5.5000, A 0.000, B 0.000, C 0.000 }
gfCNCPoint4[9322] = {X -3.5443, Y 39.9427, Z -5.5000, A 0.000, B 0.000, C 0.000 }
gfCNCPoint4[9323] = {X -3.6231, Y 39.6894, Z -5.5000, A 0.000, B 0.000, C 0.000 }
gfCNCPoint4[9324] = {X -3.6966, Y 39.4345, Z -5.5000, A 0.000, B 0.000, C 0.000 }
gfCNCPoint4[9325] = {X -4.7658, Y 35.5800, Z -5.5000, A 0.000, B 0.000, C 0.000 }
gfCNCPoint4[9326] = {X -8.0040, Y 35.6302, Z -5.5000, A 0.000, B 0.000, C 0.000 }
gfCNCPoint4[9327] = {X -8.0040, Y 35.6302, Z -2.5000, A 0.000, B 0.000, C 0.000 }
gfCNCPoint4[9328] = {X -8.0040, Y 35.6302, Z 11.0000, A 0.000, B 0.000, C 0.000 }
gfCNCPoint4[9329] = {X -7.6966, Y 17.3017, Z 11.0000, A 0.000, B 0.000, C 0.000 }
gfCNCPoint4[9330] = {X -7.6966, Y 17.3017, Z -2.5000, A 0.000, B 0.000, C 0.000 }
gfCNCPoint4[9331] = {X -7.6966, Y 17.3017, Z -5.5000, A 0.000, B 0.000, C 0.000 }
gfCNCPoint4[9332] = {X -4.2189, Y 17.3017, Z -5.5000, A 0.000, B 0.000, C 0.000 }
gfCNCPoint4[9333] = {X -3.6966, Y 13.3360, Z -5.5000, A 0.000, B 0.000, C 0.000 }
gfCNCPoint4[9334] = {X -3.6096, Y 12.8766, Z -5.5000, A 0.000, B 0.000, C 0.000 }
gfCNCPoint4[9335] = {X -3.4716, Y 12.4299, Z -5.5000, A 0.000, B 0.000, C 0.000 }
gfCNCPoint4[9336] = {X -3.0336, Y 11.5716, Z -5.5000, A 0.000, B 0.000, C 0.000 }
gfCNCPoint4[9337] = {X -2.4097, Y 10.8371, Z -5.5000, A 0.000, B 0.000, C 0.000 }
gfCNCPoint4[9338] = {X -1.6337, Y 10.2658, Z -5.5000, A 0.000, B 0.000, C 0.000 }
gfCNCPoint4[9339] = {X -1.0364, Y 9.9250, Z -5.5000, A 0.000, B 0.000, C 0.000 }
gfCNCPoint4[9340] = {X -0.1661, Y 9.5526, Z -5.5000, A 0.000, B 0.000, C 0.000 }
gfCNCPoint4[9341] = {X 0.7658, Y 9.3865, Z -5.5000, A 0.000, B 0.000, C 0.000 }
gfCNCPoint4[9342] = {X 1.7112, Y 9.4355, Z -5.5000, A 0.000, B 0.000, C 0.000 }
gfCNCPoint4[9343] = {X 2.6210, Y 9.6968, Z -5.5000, A 0.000, B 0.000, C 0.000 }
gfCNCPoint4[9344] = {X 3.4219, Y 9.3077, Z -5.5000, A 0.000, B 0.000, C 0.000 }
gfCNCPoint4[9345] = {X 4.2547, Y 8.9924, Z -5.5000, A 0.000, B 0.000, C 0.000 }
gfCNCPoint4[9346] = {X 6.1529, Y 8.3281, Z -5.5000, A 0.000, B 0.000, C 0.000 }
gfCNCPoint4[9347] = {X 8.1012, Y 7.8300, Z -5.5000, A 0.000, B 0.000, C 0.000 }
gfCNCPoint4[9348] = {X 10.0853, Y 7.5017, Z -5.5000, A 0.000, B 0.000, C 0.000 }
gfCNCPoint4[9349] = {X 12.0903, Y 7.3456, Z -5.5000, A 0.000, B 0.000, C 0.000 }
gfCNCPoint4[9350] = {X 14.1012, Y 7.3630, Z -5.5000, A 0.000, B 0.000, C 0.000 }
gfCNCPoint4[9351] = {X 16.1032, Y 7.5537, Z -5.5000, A 0.000, B 0.000, C 0.000 }
gfCNCPoint4[9352] = {X 17.9099, Y 7.8841, Z -5.5000, A 0.000, B 0.000, C 0.000 }
gfCNCPoint4[9353] = {X 19.6713, Y 8.4043, Z -5.5000, A 0.000, B 0.000, C 0.000 }
gfCNCPoint4[9354] = {X 21.3677, Y 9.1084, Z -5.5000, A 0.000, B 0.000, C 0.000 }
gfCNCPoint4[9355] = {X 22.9797, Y 9.9884, Z -5.5000, A 0.000, B 0.000, C 0.000 }
gfCNCPoint4[9356] = {X 24.4894, Y 11.0345, Z -5.5000, A 0.000, B 0.000, C 0.000 }
gfCNCPoint4[9357] = {X 25.5612, Y 11.9717, Z -5.5000, A 0.000, B 0.000, C 0.000 }
gfCNCPoint4[9358] = {X 26.5227, Y 13.0218, Z -5.5000, A 0.000, B 0.000, C 0.000 }
gfCNCPoint4[9359] = {X 27.3620, Y 14.1720, Z -5.5000, A 0.000, B 0.000, C 0.000 }
gfCNCPoint4[9360] = {X 28.0688, Y 15.4080, Z -5.5000, A 0.000, B 0.000, C 0.000 }
gfCNCPoint4[9361] = {X 28.6344, Y 16.7147, Z -5.5000, A 0.000, B 0.000, C 0.000 }
gfCNCPoint4[9362] = {X 29.1040, Y 18.3528, Z -5.5000, A 0.000, B 0.000, C 0.000 }
gfCNCPoint4[9363] = {X 29.3826, Y 20.0340, Z -5.5000, A 0.000, B 0.000, C 0.000 }
gfCNCPoint4[9364] = {X 29.4665, Y 21.7361, Z -5.5000, A 0.000, B 0.000, C 0.000 }
gfCNCPoint4[9365] = {X 29.3547, Y 23.4365, Z -5.5000, A 0.000, B 0.000, C 0.000 }
gfCNCPoint4[9366] = {X 29.0486, Y 25.1129, Z -5.5000, A 0.000, B 0.000, C 0.000 }
gfCNCPoint4[9367] = {X 28.5902, Y 26.5979, Z -5.5000, A 0.000, B 0.000, C 0.000 }
gfCNCPoint4[9368] = {X 27.9363, Y 28.0078, Z -5.5000, A 0.000, B 0.000, C 0.000 }
gfCNCPoint4[9369] = {X 27.0987, Y 29.3169, Z -5.5000, A 0.000, B 0.000, C 0.000 }
gfCNCPoint4[9370] = {X 26.0927, Y 30.5015, Z -5.5000, A 0.000, B 0.000, C 0.000 }
gfCNCPoint4[9371] = {X 24.9366, Y 31.5401, Z -5.5000, A 0.000, B 0.000, C 0.000 }
gfCNCPoint4[9372] = {X 25.1522, Y 31.5960, Z -5.5000, A 0.000, B 0.000, C 0.000 }
gfCNCPoint4[9373] = {X 25.3644, Y 31.6634, Z -5.5000, A 0.000, B 0.000, C 0.000 }
gfCNCPoint4[9374] = {X 26.0977, Y 32.0008, Z -5.5000, A 0.000, B 0.000, C 0.000 }
gfCNCPoint4[9375] = {X 26.7521, Y 32.4735, Z -5.5000, A 0.000, B 0.000, C 0.000 }
gfCNCPoint4[9376] = {X 27.3028, Y 33.0637, Z -5.5000, A 0.000, B 0.000, C 0.000 }
gfCNCPoint4[9377] = {X 27.7292, Y 33.7491, Z -5.5000, A 0.000, B 0.000, C 0.000 }
gfCNCPoint4[9378] = {X 30.7660, Y 40.0227, Z -5.5000, A 0.000, B 0.000, C 0.000 }
gfCNCPoint4[9379] = {X 31.0747, Y 40.8982, Z -5.5000, A 0.000, B 0.000, C 0.000 }
gfCNCPoint4[9380] = {X 31.1815, Y 41.8203, Z -5.5000, A 0.000, B 0.000, C 0.000 }
gfCNCPoint4[9381] = {X 31.0813, Y 42.7431, Z -5.5000, A 0.000, B 0.000, C 0.000 }
gfCNCPoint4[9382] = {X 30.7789, Y 43.6208, Z -5.5000, A 0.000, B 0.000, C 0.000 }
gfCNCPoint4[9383] = {X 30.2893, Y 44.4095, Z -5.5000, A 0.000, B 0.000, C 0.000 }
gfCNCPoint4[9384] = {X 29.6371, Y 45.0700, Z -5.5000, A 0.000, B 0.000, C 0.000 }
gfCNCPoint4[9385] = {X 29.1011, Y 45.5035, Z -5.5000, A 0.000, B 0.000, C 0.000 }
gfCNCPoint4[9386] = {X 28.4108, Y 45.9563, Z -5.5000, A 0.000, B 0.000, C 0.000 }
gfCNCPoint4[9387] = {X 27.6449, Y 46.2644, Z -5.5000, A 0.000, B 0.000, C 0.000 }
gfCNCPoint4[9388] = {X 26.8334, Y 46.4156, Z -5.5000, A 0.000, B 0.000, C 0.000 }
gfCNCPoint4[9389] = {X 26.0080, Y 46.4042, Z -5.5000, A 0.000, B 0.000, C 0.000 }
gfCNCPoint4[9390] = {X 25.2010, Y 46.2304, Z -5.5000, A 0.000, B 0.000, C 0.000 }
gfCNCPoint4[9391] = {X 23.3919, Y 47.1901, Z -5.5000, A 0.000, B 0.000, C 0.000 }
gfCNCPoint4[9392] = {X 21.5197, Y 48.0198, Z -5.5000, A 0.000, B 0.000, C 0.000 }
gfCNCPoint4[9393] = {X 19.5937, Y 48.7156, Z -5.5000, A 0.000, B 0.000, C 0.000 }
gfCNCPoint4[9394] = {X 17.6674, Y 49.2591, Z -5.5000, A 0.000, B 0.000, C 0.000 }
gfCNCPoint4[9395] = {X 15.7005, Y 49.6302, Z -5.5000, A 0.000, B 0.000, C 0.000 }
gfCNCPoint4[9396] = {X 13.7085, Y 49.8258, Z -5.5000, A 0.000, B 0.000, C 0.000 }
gfCNCPoint4[9397] = {X 11.7071, Y 49.8444, Z -5.5000, A 0.000, B 0.000, C 0.000 }
gfCNCPoint4[9398] = {X 9.7118, Y 49.6859, Z -5.5000, A 0.000, B 0.000, C 0.000 }
gfCNCPoint4[9399] = {X 7.7384, Y 49.3515, Z -5.5000, A 0.000, B 0.000, C 0.000 }
gfCNCPoint4[9400] = {X 5.8549, Y 48.8359, Z -5.5000, A 0.000, B 0.000, C 0.000 }
gfCNCPoint4[9401] = {X 4.0453, Y 48.1018, Z -5.5000, A 0.000, B 0.000, C 0.000 }
gfCNCPoint4[9402] = {X 2.3349, Y 47.1594, Z -5.5000, A 0.000, B 0.000, C 0.000 }
gfCNCPoint4[9403] = {X 0.7475, Y 46.0220, Z -5.5000, A 0.000, B 0.000, C 0.000 }
gfCNCPoint4[9404] = {X -0.3712, Y 45.0165, Z -5.5000, A 0.000, B 0.000, C 0.000 }
gfCNCPoint4[9405] = {X -1.3648, Y 43.8872, Z -5.5000, A 0.000, B 0.000, C 0.000 }
gfCNCPoint4[9406] = {X -2.2196, Y 42.6496, Z -5.5000, A 0.000, B 0.000, C 0.000 }
gfCNCPoint4[9407] = {X -2.9240, Y 41.3205, Z -5.5000, A 0.000, B 0.000, C 0.000 }
gfCNCPoint4[9408] = {X -3.4682, Y 39.9182, Z -5.5000, A 0.000, B 0.000, C 0.000 }
gfCNCPoint4[9409] = {X -3.5888, Y 39.5219, Z -5.5000, A 0.000, B 0.000, C 0.000 }
gfCNCPoint4[9410] = {X -3.6966, Y 39.1220, Z -5.5000, A 0.000, B 0.000, C 0.000 }
gfCNCPoint4[9411] = {X -4.6752, Y 35.2435, Z -5.5000, A 0.000, B 0.000, C 0.000 }
gfCNCPoint4[9412] = {X -8.0059, Y 35.2215, Z -5.5000, A 0.000, B 0.000, C 0.000 }
gfCNCPoint4[9413] = {X -8.0059, Y 35.2215, Z -2.5000, A 0.000, B 0.000, C 0.000 }
gfCNCPoint4[9414] = {X -8.0059, Y 35.2215, Z 11.0000, A 0.000, B 0.000, C 0.000 }
gfCNCPoint4[9415] = {X -7.9985, Y 34.8092, Z 11.0000, A 0.000, B 0.000, C 0.000 }
gfCNCPoint4[9416] = {X -7.9985, Y 34.8092, Z -2.5000, A 0.000, B 0.000, C 0.000 }
gfCNCPoint4[9417] = {X -7.9985, Y 34.8092, Z -5.5000, A 0.000, B 0.000, C 0.000 }
gfCNCPoint4[9418] = {X -4.8503, Y 34.9002, Z -5.5000, A 0.000, B 0.000, C 0.000 }
gfCNCPoint4[9419] = {X -3.6966, Y 31.0702, Z -5.5000, A 0.000, B 0.000, C 0.000 }
gfCNCPoint4[9420] = {X -3.6590, Y 30.9474, Z -5.5000, A 0.000, B 0.000, C 0.000 }
gfCNCPoint4[9421] = {X -3.6204, Y 30.8250, Z -5.5000, A 0.000, B 0.000, C 0.000 }
gfCNCPoint4[9422] = {X -3.4458, Y 30.3121, Z -5.5000, A 0.000, B 0.000, C 0.000 }
gfCNCPoint4[9423] = {X -3.2525, Y 29.8059, Z -5.5000, A 0.000, B 0.000, C 0.000 }
gfCNCPoint4[9424] = {X -2.6179, Y 28.4661, Z -5.5000, A 0.000, B 0.000, C 0.000 }
gfCNCPoint4[9425] = {X -1.8062, Y 27.2256, Z -5.5000, A 0.000, B 0.000, C 0.000 }
gfCNCPoint4[9426] = {X -0.8326, Y 26.1076, Z -5.5000, A 0.000, B 0.000, C 0.000 }
gfCNCPoint4[9427] = {X 0.2846, Y 25.1332, Z -5.5000, A 0.000, B 0.000, C 0.000 }
gfCNCPoint4[9428] = {X 1.5245, Y 24.3205, Z -5.5000, A 0.000, B 0.000, C 0.000 }
gfCNCPoint4[9429] = {X 1.4476, Y 24.2909, Z -5.5000, A 0.000, B 0.000, C 0.000 }
gfCNCPoint4[9430] = {X 1.3713, Y 24.2598, Z -5.5000, A 0.000, B 0.000, C 0.000 }
gfCNCPoint4[9431] = {X 0.6325, Y 23.8623, Z -5.5000, A 0.000, B 0.000, C 0.000 }
gfCNCPoint4[9432] = {X -0.0156, Y 23.3295, Z -5.5000, A 0.000, B 0.000, C 0.000 }
gfCNCPoint4[9433] = {X -0.5484, Y 22.6815, Z -5.5000, A 0.000, B 0.000, C 0.000 }
gfCNCPoint4[9434] = {X -0.9460, Y 21.9427, Z -5.5000, A 0.000, B 0.000, C 0.000 }
gfCNCPoint4[9435] = {X -3.6216, Y 15.3840, Z -5.5000, A 0.000, B 0.000, C 0.000 }
gfCNCPoint4[9436] = {X -3.6606, Y 15.2747, Z -5.5000, A 0.000, B 0.000, C 0.000 }
gfCNCPoint4[9437] = {X -3.6966, Y 15.1644, Z -5.5000, A 0.000, B 0.000, C 0.000 }
gfCNCPoint4[9438] = {X -4.8866, Y 11.3455, Z -5.5000, A 0.000, B 0.000, C 0.000 }
gfCNCPoint4[9439] = {X -7.6966, Y 11.3455, Z -5.5000, A 0.000, B 0.000, C 0.000 }
gfCNCPoint4[9440] = {X -7.6966, Y 11.3455, Z -2.5000, A 0.000, B 0.000, C 0.000 }
gfCNCPoint4[9441] = {X -7.6966, Y 11.3455, Z 11.0000, A 0.000, B 0.000, C 0.000 }
gfCNCPoint4[9442] = {X -8.0055, Y 35.1784, Z 11.0000, A 0.000, B 0.000, C 0.000 }
gfCNCPoint4[9443] = {X -8.0055, Y 35.1784, Z -2.5000, A 0.000, B 0.000, C 0.000 }
gfCNCPoint4[9444] = {X -8.0055, Y 35.1784, Z -5.5000, A 0.000, B 0.000, C 0.000 }
gfCNCPoint4[9445] = {X -4.7789, Y 35.2072, Z -5.5000, A 0.000, B 0.000, C 0.000 }
gfCNCPoint4[9446] = {X -3.6966, Y 31.3564, Z -5.5000, A 0.000, B 0.000, C 0.000 }
gfCNCPoint4[9447] = {X -3.6227, Y 31.1022, Z -5.5000, A 0.000, B 0.000, C 0.000 }
gfCNCPoint4[9448] = {X -3.5442, Y 30.8494, Z -5.5000, A 0.000, B 0.000, C 0.000 }
gfCNCPoint4[9449] = {X -3.3705, Y 30.3391, Z -5.5000, A 0.000, B 0.000, C 0.000 }
gfCNCPoint4[9450] = {X -3.1781, Y 29.8355, Z -5.5000, A 0.000, B 0.000, C 0.000 }
gfCNCPoint4[9451] = {X -2.5308, Y 28.4744, Z -5.5000, A 0.000, B 0.000, C 0.000 }
gfCNCPoint4[9452] = {X -1.6993, Y 27.2174, Z -5.5000, A 0.000, B 0.000, C 0.000 }
gfCNCPoint4[9453] = {X -0.7002, Y 26.0890, Z -5.5000, A 0.000, B 0.000, C 0.000 }
gfCNCPoint4[9454] = {X 0.4471, Y 25.1116, Z -5.5000, A 0.000, B 0.000, C 0.000 }
gfCNCPoint4[9455] = {X 1.7198, Y 24.3043, Z -5.5000, A 0.000, B 0.000, C 0.000 }
gfCNCPoint4[9456] = {X 1.5598, Y 24.2483, Z -5.5000, A 0.000, B 0.000, C 0.000 }
gfCNCPoint4[9457] = {X 1.4022, Y 24.1860, Z -5.5000, A 0.000, B 0.000, C 0.000 }
gfCNCPoint4[9458] = {X 0.6770, Y 23.7959, Z -5.5000, A 0.000, B 0.000, C 0.000 }
gfCNCPoint4[9459] = {X 0.0410, Y 23.2729, Z -5.5000, A 0.000, B 0.000, C 0.000 }
gfCNCPoint4[9460] = {X -0.4820, Y 22.6369, Z -5.5000, A 0.000, B 0.000, C 0.000 }
gfCNCPoint4[9461] = {X -0.8722, Y 21.9118, Z -5.5000, A 0.000, B 0.000, C 0.000 }
gfCNCPoint4[9462] = {X -3.5466, Y 15.3562, Z -5.5000, A 0.000, B 0.000, C 0.000 }
gfCNCPoint4[9463] = {X -3.6291, Y 15.1116, Z -5.5000, A 0.000, B 0.000, C 0.000 }
gfCNCPoint4[9464] = {X -3.6966, Y 14.8625, Z -5.5000, A 0.000, B 0.000, C 0.000 }
gfCNCPoint4[9465] = {X -4.6243, Y 10.9716, Z -5.5000, A 0.000, B 0.000, C 0.000 }
gfCNCPoint4[9466] = {X -7.6966, Y 10.9716, Z -5.5000, A 0.000, B 0.000, C 0.000 }
gfCNCPoint4[9467] = {X -7.6966, Y 10.9716, Z -2.5000, A 0.000, B 0.000, C 0.000 }
gfCNCPoint4[9468] = {X -7.6966, Y 10.9716, Z 11.0000, A 0.000, B 0.000, C 0.000 }
gfCNCPoint4[9469] = {X -8.0048, Y 35.5765, Z 11.0000, A 0.000, B 0.000, C 0.000 }
gfCNCPoint4[9470] = {X -8.0048, Y 35.5765, Z -2.5000, A 0.000, B 0.000, C 0.000 }
gfCNCPoint4[9471] = {X -8.0048, Y 35.5765, Z -5.5000, A 0.000, B 0.000, C 0.000 }
gfCNCPoint4[9472] = {X -4.7011, Y 35.5349, Z -5.5000, A 0.000, B 0.000, C 0.000 }
gfCNCPoint4[9473] = {X -3.6966, Y 31.6631, Z -5.5000, A 0.000, B 0.000, C 0.000 }
gfCNCPoint4[9474] = {X -3.5879, Y 31.2668, Z -5.5000, A 0.000, B 0.000, C 0.000 }
gfCNCPoint4[9475] = {X -3.4680, Y 30.8738, Z -5.5000, A 0.000, B 0.000, C 0.000 }
gfCNCPoint4[9476] = {X -3.2951, Y 30.3661, Z -5.5000, A 0.000, B 0.000, C 0.000 }
gfCNCPoint4[9477] = {X -3.1038, Y 29.8651, Z -5.5000, A 0.000, B 0.000, C 0.000 }
gfCNCPoint4[9478] = {X -2.4421, Y 28.4803, Z -5.5000, A 0.000, B 0.000, C 0.000 }
gfCNCPoint4[9479] = {X -1.5885, Y 27.2048, Z -5.5000, A 0.000, B 0.000, C 0.000 }
gfCNCPoint4[9480] = {X -0.5607, Y 26.0651, Z -5.5000, A 0.000, B 0.000, C 0.000 }
gfCNCPoint4[9481] = {X 0.6202, Y 25.0847, Z -5.5000, A 0.000, B 0.000, C 0.000 }
gfCNCPoint4[9482] = {X 1.9295, Y 24.2840, Z -5.5000, A 0.000, B 0.000, C 0.000 }
gfCNCPoint4[9483] = {X 1.6785, Y 24.2060, Z -5.5000, A 0.000, B 0.000, C 0.000 }
gfCNCPoint4[9484] = {X 1.4330, Y 24.1122, Z -5.5000, A 0.000, B 0.000, C 0.000 }
gfCNCPoint4[9485] = {X 0.7216, Y 23.7294, Z -5.5000, A 0.000, B 0.000, C 0.000 }
gfCNCPoint4[9486] = {X 0.0975, Y 23.2164, Z -5.5000, A 0.000, B 0.000, C 0.000 }
gfCNCPoint4[9487] = {X -0.4156, Y 22.5923, Z -5.5000, A 0.000, B 0.000, C 0.000 }
gfCNCPoint4[9488] = {X -0.7984, Y 21.8809, Z -5.5000, A 0.000, B 0.000, C 0.000 }
gfCNCPoint4[9489] = {X -3.4716, Y 15.3283, Z -5.5000, A 0.000, B 0.000, C 0.000 }
gfCNCPoint4[9490] = {X -3.6096, Y 14.8816, Z -5.5000, A 0.000, B 0.000, C 0.000 }
gfCNCPoint4[9491] = {X -3.6966, Y 14.4223, Z -5.5000, A 0.000, B 0.000, C 0.000 }
gfCNCPoint4[9492] = {X -4.2189, Y 10.4565, Z -5.5000, A 0.000, B 0.000, C 0.000 }
gfCNCPoint4[9493] = {X -7.6966, Y 10.4565, Z -5.5000, A 0.000, B 0.000, C 0.000 }
gfCNCPoint4[9494] = {X -7.6966, Y 10.4565, Z -2.5000, A 0.000, B 0.000, C 0.000 }
gfCNCPoint4[9495] = {X -7.6966, Y 10.4565, Z 11.0000, A 0.000, B 0.000, C 0.000 }
gfCNCPoint4[9496] = {X -7.9942, Y 36.0109, Z 11.0000, A 0.000, B 0.000, C 0.000 }
gfCNCPoint4[9497] = {X -7.9942, Y 36.0109, Z -2.5000, A 0.000, B 0.000, C 0.000 }
gfCNCPoint4[9498] = {X -7.9942, Y 36.0109, Z -5.5000, A 0.000, B 0.000, C 0.000 }
gfCNCPoint4[9499] = {X -4.6153, Y 35.8889, Z -5.5000, A 0.000, B 0.000, C 0.000 }
gfCNCPoint4[9500] = {X -3.6966, Y 31.9958, Z -5.5000, A 0.000, B 0.000, C 0.000 }
gfCNCPoint4[9501] = {X -3.5550, Y 31.4440, Z -5.5000, A 0.000, B 0.000, C 0.000 }
gfCNCPoint4[9502] = {X -3.3918, Y 30.8982, Z -5.5000, A 0.000, B 0.000, C 0.000 }
gfCNCPoint4[9503] = {X -3.2198, Y 30.3931, Z -5.5000, A 0.000, B 0.000, C 0.000 }
gfCNCPoint4[9504] = {X -3.0294, Y 29.8946, Z -5.5000, A 0.000, B 0.000, C 0.000 }
gfCNCPoint4[9505] = {X -2.3514, Y 28.4828, Z -5.5000, A 0.000, B 0.000, C 0.000 }
gfCNCPoint4[9506] = {X -1.4725, Y 27.1866, Z -5.5000, A 0.000, B 0.000, C 0.000 }
gfCNCPoint4[9507] = {X -0.4118, Y 26.0342, Z -5.5000, A 0.000, B 0.000, C 0.000 }
gfCNCPoint4[9508] = {X 0.8072, Y 25.0510, Z -5.5000, A 0.000, B 0.000, C 0.000 }
gfCNCPoint4[9509] = {X 2.1580, Y 24.2585, Z -5.5000, A 0.000, B 0.000, C 0.000 }
gfCNCPoint4[9510] = {X 1.8060, Y 24.1640, Z -5.5000, A 0.000, B 0.000, C 0.000 }
gfCNCPoint4[9511] = {X 1.4639, Y 24.0384, Z -5.5000, A 0.000, B 0.000, C 0.000 }
gfCNCPoint4[9512] = {X 0.7662, Y 23.6630, Z -5.5000, A 0.000, B 0.000, C 0.000 }
gfCNCPoint4[9513] = {X 0.1541, Y 23.1598, Z -5.5000, A 0.000, B 0.000, C 0.000 }
gfCNCPoint4[9514] = {X -0.3491, Y 22.5478, Z -5.5000, A 0.000, B 0.000, C 0.000 }
gfCNCPoint4[9515] = {X -0.7246, Y 21.8500, Z -5.5000, A 0.000, B 0.000, C 0.000 }
gfCNCPoint4[9516] = {X -3.3966, Y 15.3004, Z -5.5000, A 0.000, B 0.000, C 0.000 }
gfCNCPoint4[9517] = {X -3.6236, Y 14.3619, Z -5.5000, A 0.000, B 0.000, C 0.000 }
gfCNCPoint4[9518] = {X -3.6236, Y 13.3963, Z -5.5000, A 0.000, B 0.000, C 0.000 }
gfCNCPoint4[9519] = {X -3.3966, Y 12.4578, Z -5.5000, A 0.000, B 0.000, C 0.000 }
gfCNCPoint4[9520] = {X -2.9670, Y 11.6160, Z -5.5000, A 0.000, B 0.000, C 0.000 }
gfCNCPoint4[9521] = {X -2.3552, Y 10.8956, Z -5.5000, A 0.000, B 0.000, C 0.000 }
gfCNCPoint4[9522] = {X -1.5940, Y 10.3353, Z -5.5000, A 0.000, B 0.000, C 0.000 }
gfCNCPoint4[9523] = {X -0.9967, Y 9.9945, Z -5.5000, A 0.000, B 0.000, C 0.000 }
gfCNCPoint4[9524] = {X -0.1687, Y 9.6370, Z -5.5000, A 0.000, B 0.000, C 0.000 }
gfCNCPoint4[9525] = {X 0.7176, Y 9.4701, Z -5.5000, A 0.000, B 0.000, C 0.000 }
gfCNCPoint4[9526] = {X 1.6189, Y 9.5019, Z -5.5000, A 0.000, B 0.000, C 0.000 }
gfCNCPoint4[9527] = {X 2.4913, Y 9.7311, Z -5.5000, A 0.000, B 0.000, C 0.000 }
gfCNCPoint4[9528] = {X 2.5586, Y 9.7577, Z -5.5000, A 0.000, B 0.000, C 0.000 }
gfCNCPoint4[9529] = {X 2.6255, Y 9.7855, Z -5.5000, A 0.000, B 0.000, C 0.000 }
gfCNCPoint4[9530] = {X 3.4372, Y 9.3883, Z -5.5000, A 0.000, B 0.000, C 0.000 }
gfCNCPoint4[9531] = {X 4.2820, Y 9.0676, Z -5.5000, A 0.000, B 0.000, C 0.000 }
gfCNCPoint4[9532] = {X 6.1741, Y 8.4053, Z -5.5000, A 0.000, B 0.000, C 0.000 }
gfCNCPoint4[9533] = {X 8.1162, Y 7.9086, Z -5.5000, A 0.000, B 0.000, C 0.000 }
gfCNCPoint4[9534] = {X 10.0939, Y 7.5812, Z -5.5000, A 0.000, B 0.000, C 0.000 }
gfCNCPoint4[9535] = {X 12.0925, Y 7.4256, Z -5.5000, A 0.000, B 0.000, C 0.000 }
gfCNCPoint4[9536] = {X 14.0970, Y 7.4429, Z -5.5000, A 0.000, B 0.000, C 0.000 }
gfCNCPoint4[9537] = {X 16.0926, Y 7.6330, Z -5.5000, A 0.000, B 0.000, C 0.000 }
gfCNCPoint4[9538] = {X 17.8910, Y 7.9618, Z -5.5000, A 0.000, B 0.000, C 0.000 }
gfCNCPoint4[9539] = {X 19.6444, Y 8.4796, Z -5.5000, A 0.000, B 0.000, C 0.000 }
gfCNCPoint4[9540] = {X 21.3330, Y 9.1804, Z -5.5000, A 0.000, B 0.000, C 0.000 }
gfCNCPoint4[9541] = {X 22.9377, Y 10.0564, Z -5.5000, A 0.000, B 0.000, C 0.000 }
gfCNCPoint4[9542] = {X 24.4404, Y 11.0977, Z -5.5000, A 0.000, B 0.000, C 0.000 }
gfCNCPoint4[9543] = {X 25.5054, Y 12.0290, Z -5.5000, A 0.000, B 0.000, C 0.000 }
gfCNCPoint4[9544] = {X 26.4608, Y 13.0725, Z -5.5000, A 0.000, B 0.000, C 0.000 }
gfCNCPoint4[9545] = {X 27.2947, Y 14.2153, Z -5.5000, A 0.000, B 0.000, C 0.000 }
gfCNCPoint4[9546] = {X 27.9971, Y 15.4434, Z -5.5000, A 0.000, B 0.000, C 0.000 }
gfCNCPoint4[9547] = {X 28.5591, Y 16.7417, Z -5.5000, A 0.000, B 0.000, C 0.000 }
gfCNCPoint4[9548] = {X 29.0260, Y 18.3709, Z -5.5000, A 0.000, B 0.000, C 0.000 }
gfCNCPoint4[9549] = {X 29.3031, Y 20.0430, Z -5.5000, A 0.000, B 0.000, C 0.000 }
gfCNCPoint4[9550] = {X 29.3865, Y 21.7358, Z -5.5000, A 0.000, B 0.000, C 0.000 }
gfCNCPoint4[9551] = {X 29.2753, Y 23.4270, Z -5.5000, A 0.000, B 0.000, C 0.000 }
gfCNCPoint4[9552] = {X 28.9708, Y 25.0942, Z -5.5000, A 0.000, B 0.000, C 0.000 }
gfCNCPoint4[9553] = {X 28.5031, Y 26.6013, Z -5.5000, A 0.000, B 0.000, C 0.000 }
gfCNCPoint4[9554] = {X 27.8327, Y 28.0298, Z -5.5000, A 0.000, B 0.000, C 0.000 }
gfCNCPoint4[9555] = {X 26.9723, Y 29.3525, Z -5.5000, A 0.000, B 0.000, C 0.000 }
gfCNCPoint4[9556] = {X 25.9382, Y 30.5444, Z -5.5000, A 0.000, B 0.000, C 0.000 }
gfCNCPoint4[9557] = {X 24.7501, Y 31.5829, Z -5.5000, A 0.000, B 0.000, C 0.000 }
gfCNCPoint4[9558] = {X 25.0471, Y 31.6500, Z -5.5000, A 0.000, B 0.000, C 0.000 }
gfCNCPoint4[9559] = {X 25.3382, Y 31.7390, Z -5.5000, A 0.000, B 0.000, C 0.000 }
gfCNCPoint4[9560] = {X 26.0574, Y 32.0699, Z -5.5000, A 0.000, B 0.000, C 0.000 }
gfCNCPoint4[9561] = {X 26.6991, Y 32.5335, Z -5.5000, A 0.000, B 0.000, C 0.000 }
gfCNCPoint4[9562] = {X 27.2393, Y 33.1123, Z -5.5000, A 0.000, B 0.000, C 0.000 }
gfCNCPoint4[9563] = {X 27.6575, Y 33.7845, Z -5.5000, A 0.000, B 0.000, C 0.000 }
gfCNCPoint4[9564] = {X 30.6940, Y 40.0576, Z -5.5000, A 0.000, B 0.000, C 0.000 }
gfCNCPoint4[9565] = {X 30.9967, Y 40.9162, Z -5.5000, A 0.000, B 0.000, C 0.000 }
gfCNCPoint4[9566] = {X 31.1015, Y 41.8206, Z -5.5000, A 0.000, B 0.000, C 0.000 }
gfCNCPoint4[9567] = {X 31.0032, Y 42.7257, Z -5.5000, A 0.000, B 0.000, C 0.000 }
gfCNCPoint4[9568] = {X 30.7066, Y 43.5864, Z -5.5000, A 0.000, B 0.000, C 0.000 }
gfCNCPoint4[9569] = {X 30.2265, Y 44.3600, Z -5.5000, A 0.000, B 0.000, C 0.000 }
gfCNCPoint4[9570] = {X 29.5868, Y 45.0078, Z -5.5000, A 0.000, B 0.000, C 0.000 }
gfCNCPoint4[9571] = {X 29.0508, Y 45.4413, Z -5.5000, A 0.000, B 0.000, C 0.000 }
gfCNCPoint4[9572] = {X 28.3675, Y 45.8887, Z -5.5000, A 0.000, B 0.000, C 0.000 }
gfCNCPoint4[9573] = {X 27.6090, Y 46.1915, Z -5.5000, A 0.000, B 0.000, C 0.000 }
gfCNCPoint4[9574] = {X 26.8055, Y 46.3377, Z -5.5000, A 0.000, B 0.000, C 0.000 }
gfCNCPoint4[9575] = {X 25.9889, Y 46.3214, Z -5.5000, A 0.000, B 0.000, C 0.000 }
gfCNCPoint4[9576] = {X 25.1919, Y 46.1433, Z -5.5000, A 0.000, B 0.000, C 0.000 }
gfCNCPoint4[9577] = {X 23.3782, Y 47.1078, Z -5.5000, A 0.000, B 0.000, C 0.000 }
gfCNCPoint4[9578] = {X 21.5007, Y 47.9413, Z -5.5000, A 0.000, B 0.000, C 0.000 }
gfCNCPoint4[9579] = {X 19.5689, Y 48.6395, Z -5.5000, A 0.000, B 0.000, C 0.000 }
gfCNCPoint4[9580] = {X 17.6493, Y 49.1812, Z -5.5000, A 0.000, B 0.000, C 0.000 }
gfCNCPoint4[9581] = {X 15.6893, Y 49.5510, Z -5.5000, A 0.000, B 0.000, C 0.000 }
gfCNCPoint4[9582] = {X 13.7043, Y 49.7459, Z -5.5000, A 0.000, B 0.000, C 0.000 }
gfCNCPoint4[9583] = {X 11.7099, Y 49.7645, Z -5.5000, A 0.000, B 0.000, C 0.000 }
gfCNCPoint4[9584] = {X 9.7216, Y 49.6065, Z -5.5000, A 0.000, B 0.000, C 0.000 }
gfCNCPoint4[9585] = {X 7.7551, Y 49.2733, Z -5.5000, A 0.000, B 0.000, C 0.000 }
gfCNCPoint4[9586] = {X 5.8806, Y 48.7601, Z -5.5000, A 0.000, B 0.000, C 0.000 }
gfCNCPoint4[9587] = {X 4.0797, Y 48.0295, Z -5.5000, A 0.000, B 0.000, C 0.000 }
gfCNCPoint4[9588] = {X 2.3774, Y 47.0917, Z -5.5000, A 0.000, B 0.000, C 0.000 }
gfCNCPoint4[9589] = {X 0.7977, Y 45.9597, Z -5.5000, A 0.000, B 0.000, C 0.000 }
gfCNCPoint4[9590] = {X -0.3142, Y 44.9604, Z -5.5000, A 0.000, B 0.000, C 0.000 }
gfCNCPoint4[9591] = {X -1.3016, Y 43.8381, Z -5.5000, A 0.000, B 0.000, C 0.000 }
gfCNCPoint4[9592] = {X -2.1512, Y 42.6081, Z -5.5000, A 0.000, B 0.000, C 0.000 }
gfCNCPoint4[9593] = {X -2.8512, Y 41.2873, Z -5.5000, A 0.000, B 0.000, C 0.000 }
gfCNCPoint4[9594] = {X -3.3920, Y 39.8937, Z -5.5000, A 0.000, B 0.000, C 0.000 }
gfCNCPoint4[9595] = {X -3.5570, Y 39.3388, Z -5.5000, A 0.000, B 0.000, C 0.000 }
gfCNCPoint4[9596] = {X -3.6966, Y 38.7771, Z -5.5000, A 0.000, B 0.000, C 0.000 }
gfCNCPoint4[9597] = {X -4.5733, Y 34.8743, Z -5.5000, A 0.000, B 0.000, C 0.000 }
gfCNCPoint4[9598] = {X -7.9973, Y 34.7677, Z -5.5000, A 0.000, B 0.000, C 0.000 }
gfCNCPoint4[9599] = {X -7.9973, Y 34.7677, Z -2.5000, A 0.000, B 0.000, C 0.000 }
gfCNCPoint4[9600] = {X -7.9973, Y 34.7677, Z 11.0000, A 0.000, B 0.000, C 0.000 }
gfCNCPoint4[9601] = {X -7.9705, Y 36.4928, Z 11.0000, A 0.000, B 0.000, C 0.000 }
gfCNCPoint4[9602] = {X -7.9705, Y 36.4928, Z -2.5000, A 0.000, B 0.000, C 0.000 }
gfCNCPoint4[9603] = {X -7.9705, Y 36.4928, Z -5.5000, A 0.000, B 0.000, C 0.000 }
gfCNCPoint4[9604] = {X -4.5190, Y 36.2779, Z -5.5000, A 0.000, B 0.000, C 0.000 }
gfCNCPoint4[9605] = {X -3.6966, Y 32.3634, Z -5.5000, A 0.000, B 0.000, C 0.000 }
gfCNCPoint4[9606] = {X -3.5247, Y 31.6381, Z -5.5000, A 0.000, B 0.000, C 0.000 }
gfCNCPoint4[9607] = {X -3.3157, Y 30.9226, Z -5.5000, A 0.000, B 0.000, C 0.000 }
gfCNCPoint4[9608] = {X -3.1443, Y 30.4194, Z -5.5000, A 0.000, B 0.000, C 0.000 }
gfCNCPoint4[9609] = {X -2.9546, Y 29.9228, Z -5.5000, A 0.000, B 0.000, C 0.000 }
gfCNCPoint4[9610] = {X -2.3886, Y 28.7126, Z -5.5000, A 0.000, B 0.000, C 0.000 }
gfCNCPoint4[9611] = {X -1.6737, Y 27.5841, Z -5.5000, A 0.000, B 0.000, C 0.000 }
gfCNCPoint4[9612] = {X -0.8213, Y 26.5554, Z -5.5000, A 0.000, B 0.000, C 0.000 }
gfCNCPoint4[9613] = {X 0.1548, Y 25.6433, Z -5.5000, A 0.000, B 0.000, C 0.000 }
gfCNCPoint4[9614] = {X 1.2388, Y 24.8624, Z -5.5000, A 0.000, B 0.000, C 0.000 }
gfCNCPoint4[9615] = {X 2.4131, Y 24.2254, Z -5.5000, A 0.000, B 0.000, C 0.000 }
gfCNCPoint4[9616] = {X 1.9461, Y 24.1225, Z -5.5000, A 0.000, B 0.000, C 0.000 }
gfCNCPoint4[9617] = {X 1.4948, Y 23.9646, Z -5.5000, A 0.000, B 0.000, C 0.000 }
gfCNCPoint4[9618] = {X 0.8034, Y 23.5917, Z -5.5000, A 0.000, B 0.000, C 0.000 }
gfCNCPoint4[9619] = {X 0.1983, Y 23.0908, Z -5.5000, A 0.000, B 0.000, C 0.000 }
gfCNCPoint4[9620] = {X -0.2973, Y 22.4813, Z -5.5000, A 0.000, B 0.000, C 0.000 }
gfCNCPoint4[9621] = {X -0.6642, Y 21.7867, Z -5.5000, A 0.000, B 0.000, C 0.000 }
gfCNCPoint4[9622] = {X -3.2754, Y 15.3911, Z -5.5000, A 0.000, B 0.000, C 0.000 }
gfCNCPoint4[9623] = {X -3.2990, Y 15.3320, Z -5.5000, A 0.000, B 0.000, C 0.000 }
gfCNCPoint4[9624] = {X -3.3217, Y 15.2726, Z -5.5000, A 0.000, B 0.000, C 0.000 }
gfCNCPoint4[9625] = {X -3.5441, Y 14.3524, Z -5.5000, A 0.000, B 0.000, C 0.000 }
gfCNCPoint4[9626] = {X -3.5441, Y 13.4058, Z -5.5000, A 0.000, B 0.000, C 0.000 }
gfCNCPoint4[9627] = {X -3.3217, Y 12.4857, Z -5.5000, A 0.000, B 0.000, C 0.000 }
gfCNCPoint4[9628] = {X -2.9004, Y 11.6603, Z -5.5000, A 0.000, B 0.000, C 0.000 }
gfCNCPoint4[9629] = {X -2.3006, Y 10.9541, Z -5.5000, A 0.000, B 0.000, C 0.000 }
gfCNCPoint4[9630] = {X -1.5544, Y 10.4048, Z -5.5000, A 0.000, B 0.000, C 0.000 }
gfCNCPoint4[9631] = {X -0.9063, Y 10.0355, Z -5.5000, A 0.000, B 0.000, C 0.000 }
gfCNCPoint4[9632] = {X -0.1035, Y 9.7009, Z -5.5000, A 0.000, B 0.000, C 0.000 }
gfCNCPoint4[9633] = {X 0.7527, Y 9.5477, Z -5.5000, A 0.000, B 0.000, C 0.000 }
gfCNCPoint4[9634] = {X 1.6217, Y 9.5832, Z -5.5000, A 0.000, B 0.000, C 0.000 }
gfCNCPoint4[9635] = {X 2.4625, Y 9.8057, Z -5.5000, A 0.000, B 0.000, C 0.000 }
gfCNCPoint4[9636] = {X 2.5465, Y 9.8392, Z -5.5000, A 0.000, B 0.000, C 0.000 }
gfCNCPoint4[9637] = {X 2.6297, Y 9.8745, Z -5.5000, A 0.000, B 0.000, C 0.000 }
gfCNCPoint4[9638] = {X 3.4578, Y 9.4661, Z -5.5000, A 0.000, B 0.000, C 0.000 }
gfCNCPoint4[9639] = {X 4.3209, Y 9.1382, Z -5.5000, A 0.000, B 0.000, C 0.000 }
gfCNCPoint4[9640] = {X 6.2051, Y 8.4795, Z -5.5000, A 0.000, B 0.000, C 0.000 }
gfCNCPoint4[9641] = {X 8.1391, Y 7.9855, Z -5.5000, A 0.000, B 0.000, C 0.000 }
gfCNCPoint4[9642] = {X 10.1085, Y 7.6600, Z -5.5000, A 0.000, B 0.000, C 0.000 }
gfCNCPoint4[9643] = {X 12.0985, Y 7.5054, Z -5.5000, A 0.000, B 0.000, C 0.000 }
gfCNCPoint4[9644] = {X 14.0945, Y 7.5229, Z -5.5000, A 0.000, B 0.000, C 0.000 }
gfCNCPoint4[9645] = {X 16.0816, Y 7.7122, Z -5.5000, A 0.000, B 0.000, C 0.000 }
gfCNCPoint4[9646] = {X 16.4822, Y 7.7686, Z -5.5000, A 0.000, B 0.000, C 0.000 }
gfCNCPoint4[9647] = {X 18.1859, Y 8.1176, Z -5.5000, A 0.000, B 0.000, C 0.000 }
gfCNCPoint4[9648] = {X 19.8454, Y 8.6375, Z -5.5000, A 0.000, B 0.000, C 0.000 }
gfCNCPoint4[9649] = {X 21.4437, Y 9.3231, Z -5.5000, A 0.000, B 0.000, C 0.000 }
gfCNCPoint4[9650] = {X 22.9643, Y 10.1671, Z -5.5000, A 0.000, B 0.000, C 0.000 }
gfCNCPoint4[9651] = {X 24.3914, Y 11.1610, Z -5.5000, A 0.000, B 0.000, C 0.000 }
gfCNCPoint4[9652] = {X 25.4496, Y 12.0863, Z -5.5000, A 0.000, B 0.000, C 0.000 }
gfCNCPoint4[9653] = {X 26.3988, Y 13.1231, Z -5.5000, A 0.000, B 0.000, C 0.000 }
gfCNCPoint4[9654] = {X 27.2274, Y 14.2585, Z -5.5000, A 0.000, B 0.000, C 0.000 }
gfCNCPoint4[9655] = {X 27.9253, Y 15.4788, Z -5.5000, A 0.000, B 0.000, C 0.000 }
gfCNCPoint4[9656] = {X 28.4838, Y 16.7687, Z -5.5000, A 0.000, B 0.000, C 0.000 }
gfCNCPoint4[9657] = {X 28.9482, Y 18.3893, Z -5.5000, A 0.000, B 0.000, C 0.000 }
gfCNCPoint4[9658] = {X 29.2236, Y 20.0524, Z -5.5000, A 0.000, B 0.000, C 0.000 }
gfCNCPoint4[9659] = {X 29.3065, Y 21.7361, Z -5.5000, A 0.000, B 0.000, C 0.000 }
gfCNCPoint4[9660] = {X 29.1957, Y 23.4182, Z -5.5000, A 0.000, B 0.000, C 0.000 }
gfCNCPoint4[9661] = {X 28.8928, Y 25.0766, Z -5.5000, A 0.000, B 0.000, C 0.000 }
gfCNCPoint4[9662] = {X 28.4147, Y 26.6079, Z -5.5000, A 0.000, B 0.000, C 0.000 }
gfCNCPoint4[9663] = {X 27.7258, Y 28.0568, Z -5.5000, A 0.000, B 0.000, C 0.000 }
gfCNCPoint4[9664] = {X 26.8400, Y 29.3943, Z -5.5000, A 0.000, B 0.000, C 0.000 }
gfCNCPoint4[9665] = {X 25.7747, Y 30.5938, Z -5.5000, A 0.000, B 0.000, C 0.000 }
gfCNCPoint4[9666] = {X 24.5512, Y 31.6315, Z -5.5000, A 0.000, B 0.000, C 0.000 }
gfCNCPoint4[9667] = {X 24.9361, Y 31.7044, Z -5.5000, A 0.000, B 0.000, C 0.000 }
gfCNCPoint4[9668] = {X 25.3120, Y 31.8146, Z -5.5000, A 0.000, B 0.000, C 0.000 }
gfCNCPoint4[9669] = {X 26.0245, Y 32.1433, Z -5.5000, A 0.000, B 0.000, C 0.000 }
gfCNCPoint4[9670] = {X 26.6591, Y 32.6049, Z -5.5000, A 0.000, B 0.000, C 0.000 }
gfCNCPoint4[9671] = {X 27.1913, Y 33.1814, Z -5.5000, A 0.000, B 0.000, C 0.000 }
gfCNCPoint4[9672] = {X 27.6008, Y 33.8508, Z -5.5000, A 0.000, B 0.000, C 0.000 }
gfCNCPoint4[9673] = {X 30.6220, Y 40.0925, Z -5.5000, A 0.000, B 0.000, C 0.000 }
gfCNCPoint4[9674] = {X 30.9188, Y 40.9342, Z -5.5000, A 0.000, B 0.000, C 0.000 }
gfCNCPoint4[9675] = {X 31.0215, Y 41.8209, Z -5.5000, A 0.000, B 0.000, C 0.000 }
gfCNCPoint4[9676] = {X 30.9251, Y 42.7082, Z -5.5000, A 0.000, B 0.000, C 0.000 }
gfCNCPoint4[9677] = {X 30.6343, Y 43.5521, Z -5.5000, A 0.000, B 0.000, C 0.000 }
gfCNCPoint4[9678] = {X 30.1637, Y 44.3105, Z -5.5000, A 0.000, B 0.000, C 0.000 }
gfCNCPoint4[9679] = {X 29.5365, Y 44.9456, Z -5.5000, A 0.000, B 0.000, C 0.000 }
gfCNCPoint4[9680] = {X 29.0005, Y 45.3790, Z -5.5000, A 0.000, B 0.000, C 0.000 }
gfCNCPoint4[9681] = {X 28.3242, Y 45.8210, Z -5.5000, A 0.000, B 0.000, C 0.000 }
gfCNCPoint4[9682] = {X 27.5731, Y 46.1185, Z -5.5000, A 0.000, B 0.000, C 0.000 }
gfCNCPoint4[9683] = {X 26.7777, Y 46.2596, Z -5.5000, A 0.000, B 0.000, C 0.000 }
gfCNCPoint4[9684] = {X 25.9701, Y 46.2384, Z -5.5000, A 0.000, B 0.000, C 0.000 }
gfCNCPoint4[9685] = {X 25.1831, Y 46.0559, Z -5.5000, A 0.000, B 0.000, C 0.000 }
gfCNCPoint4[9686] = {X 25.1073, Y 46.0997, Z -5.5000, A 0.000, B 0.000, C 0.000 }
